   "HMI_DB".Drives.CU_U1.STW1.Bit00 := "DB_CU_U1".TelOut.CU_STW1.%X0;
   "HMI_DB".Drives.CU_U1.STW1.Bit01 := "DB_CU_U1".TelOut.CU_STW1.%X1;
   "HMI_DB".Drives.CU_U1.STW1.Bit02 := "DB_CU_U1".TelOut.CU_STW1.%X2;
   "HMI_DB".Drives.CU_U1.STW1.Bit03 := "DB_CU_U1".TelOut.CU_STW1.%X3;
   "HMI_DB".Drives.CU_U1.STW1.Bit04 := "DB_CU_U1".TelOut.CU_STW1.%X4;
   "HMI_DB".Drives.CU_U1.STW1.Bit05 := "DB_CU_U1".TelOut.CU_STW1.%X5;
   "HMI_DB".Drives.CU_U1.STW1.Bit06 := "DB_CU_U1".TelOut.CU_STW1.%X6;
   "HMI_DB".Drives.CU_U1.STW1.FaultAcknowledge := "DB_CU_U1".TelOut.CU_STW1.%X7;
   "HMI_DB".Drives.CU_U1.STW1.Bit08 := "DB_CU_U1".TelOut.CU_STW1.%X8;
   "HMI_DB".Drives.CU_U1.STW1.Bit09 := "DB_CU_U1".TelOut.CU_STW1.%X9;
   "HMI_DB".Drives.CU_U1.STW1.RemoteControlByPLC := "DB_CU_U1".TelOut.CU_STW1.%X10;
   "HMI_DB".Drives.CU_U1.STW1.Bit11 := "DB_CU_U1".TelOut.CU_STW1.%X11;
   "HMI_DB".Drives.CU_U1.STW1.Bit12 := "DB_CU_U1".TelOut.CU_STW1.%X12;
   "HMI_DB".Drives.CU_U1.STW1.Bit13 := "DB_CU_U1".TelOut.CU_STW1.%X13;
   "HMI_DB".Drives.CU_U1.STW1.Bit14 := "DB_CU_U1".TelOut.CU_STW1.%X14;
   "HMI_DB".Drives.CU_U1.STW1.Bit15 := "DB_CU_U1".TelOut.CU_STW1.%X15;


   // ============================================================
   // 6. CU_ZSW1 bits, CU -> PLC
   // ============================================================

   "HMI_DB".Drives.CU_U1.ZSW1.ReadyToSwitchOn := "DB_CU_U1".TelIn.CU_ZSW1.%X0;
   "HMI_DB".Drives.CU_U1.ZSW1.ReadyToOperate := "DB_CU_U1".TelIn.CU_ZSW1.%X1;
   "HMI_DB".Drives.CU_U1.ZSW1.OperationEnabled := "DB_CU_U1".TelIn.CU_ZSW1.%X2;
   "HMI_DB".Drives.CU_U1.ZSW1.FaultActive := "DB_CU_U1".TelIn.CU_ZSW1.%X3;
   "HMI_DB".Drives.CU_U1.ZSW1.NoCoastStopActive := "DB_CU_U1".TelIn.CU_ZSW1.%X4;
   "HMI_DB".Drives.CU_U1.ZSW1.NoQuickStopActive := "DB_CU_U1".TelIn.CU_ZSW1.%X5;
   "HMI_DB".Drives.CU_U1.ZSW1.SwitchingOnInhibit := "DB_CU_U1".TelIn.CU_ZSW1.%X6;
   "HMI_DB".Drives.CU_U1.ZSW1.WarningActive := "DB_CU_U1".TelIn.CU_ZSW1.%X7;
   "HMI_DB".Drives.CU_U1.ZSW1.Bit08 := "DB_CU_U1".TelIn.CU_ZSW1.%X8;
   "HMI_DB".Drives.CU_U1.ZSW1.ControlRequested := "DB_CU_U1".TelIn.CU_ZSW1.%X9;
   "HMI_DB".Drives.CU_U1.ZSW1.Bit10 := "DB_CU_U1".TelIn.CU_ZSW1.%X10;
   "HMI_DB".Drives.CU_U1.ZSW1.Bit11 := "DB_CU_U1".TelIn.CU_ZSW1.%X11;
   "HMI_DB".Drives.CU_U1.ZSW1.Bit12 := "DB_CU_U1".TelIn.CU_ZSW1.%X12;
   "HMI_DB".Drives.CU_U1.ZSW1.Bit13 := "DB_CU_U1".TelIn.CU_ZSW1.%X13;
   "HMI_DB".Drives.CU_U1.ZSW1.Bit14 := "DB_CU_U1".TelIn.CU_ZSW1.%X14;
   "HMI_DB".Drives.CU_U1.ZSW1.Bit15 := "DB_CU_U1".TelIn.CU_ZSW1.%X15;
END_REGION
END_FUNCTION

FUNCTION "FC_Drives_HMI_Alarms" : Void   // FC53, LAD
TITLE = Формування слів аварій (Faults) ПЧ для HMI
{ S7_Optimized_Access := 'TRUE' }
VERSION : 0.1
BEGIN

REGION Network 2 (SCL): Формування слів аварій для HMI - ПЧ 1UZ1
   // ============================================================
   // 1. FaultsWord1
   // ============================================================

   "HMI_DB".Drives.Drive_1UZ1.Faults.FaultsWord1.%X0 := "DB_Drive_1UZ1".Status.%X4 AND ("DB_Drive_1UZ1".FaultCode = W#16#03E8); // F01000
   "HMI_DB".Drives.Drive_1UZ1.Faults.FaultsWord1.%X1 := "DB_Drive_1UZ1".Status.%X4 AND ("DB_Drive_1UZ1".FaultCode = W#16#03E9); // F01001
   "HMI_DB".Drives.Drive_1UZ1.Faults.FaultsWord1.%X2 := "DB_Drive_1UZ1".Status.%X4 AND ("DB_Drive_1UZ1".FaultCode = W#16#03F7); // F01015
   "HMI_DB".Drives.Drive_1UZ1.Faults.FaultsWord1.%X3 := "DB_Drive_1UZ1".Status.%X4 AND ("DB_Drive_1UZ1".FaultCode = W#16#0409); // F01033
   "HMI_DB".Drives.Drive_1UZ1.Faults.FaultsWord1.%X4 := "DB_Drive_1UZ1".Status.%X4 AND ("DB_Drive_1UZ1".FaultCode = W#16#040A); // F01034
   "HMI_DB".Drives.Drive_1UZ1.Faults.FaultsWord1.%X5 := "DB_Drive_1UZ1".Status.%X4 AND ("DB_Drive_1UZ1".FaultCode = W#16#0410); // F01040
   "HMI_DB".Drives.Drive_1UZ1.Faults.FaultsWord1.%X6 := "DB_Drive_1UZ1".Status.%X4 AND ("DB_Drive_1UZ1".FaultCode = W#16#0414); // F01044
   "HMI_DB".Drives.Drive_1UZ1.Faults.FaultsWord1.%X7 := "DB_Drive_1UZ1".Status.%X4 AND ("DB_Drive_1UZ1".FaultCode = W#16#041E); // F01054
   "HMI_DB".Drives.Drive_1UZ1.Faults.FaultsWord1.%X8 := "DB_Drive_1UZ1".Status.%X4 AND ("DB_Drive_1UZ1".FaultCode = W#16#0451); // F01105
   "HMI_DB".Drives.Drive_1UZ1.Faults.FaultsWord1.%X9 := "DB_Drive_1UZ1".Status.%X4 AND ("DB_Drive_1UZ1".FaultCode = W#16#0462); // F01122
   "HMI_DB".Drives.Drive_1UZ1.Faults.FaultsWord1.%X10 := "DB_Drive_1UZ1".Status.%X4 AND ("DB_Drive_1UZ1".FaultCode = W#16#04B5); // F01205
   "HMI_DB".Drives.Drive_1UZ1.Faults.FaultsWord1.%X11 := "DB_Drive_1UZ1".Status.%X4 AND ("DB_Drive_1UZ1".FaultCode = W#16#04E2); // F01250
   "HMI_DB".Drives.Drive_1UZ1.Faults.FaultsWord1.%X12 := "DB_Drive_1UZ1".Status.%X4 AND ("DB_Drive_1UZ1".FaultCode = W#16#05E8); // F01512
   "HMI_DB".Drives.Drive_1UZ1.Faults.FaultsWord1.%X13 := "DB_Drive_1UZ1".Status.%X4 AND ("DB_Drive_1UZ1".FaultCode = W#16#0640); // F01600
   "HMI_DB".Drives.Drive_1UZ1.Faults.FaultsWord1.%X14 := "DB_Drive_1UZ1".Status.%X4 AND ("DB_Drive_1UZ1".FaultCode = W#16#0659); // F01625
   "HMI_DB".Drives.Drive_1UZ1.Faults.FaultsWord1.%X15 := "DB_Drive_1UZ1".Status.%X4 AND ("DB_Drive_1UZ1".FaultCode = W#16#0672); // F01650


   // ============================================================
   // 2. FaultsWord2
   // ============================================================

   "HMI_DB".Drives.Drive_1UZ1.Faults.FaultsWord2.%X0 := "DB_Drive_1UZ1".Status.%X4 AND ("DB_Drive_1UZ1".FaultCode = W#16#067B); // F01659
   "HMI_DB".Drives.Drive_1UZ1.Faults.FaultsWord2.%X1 := "DB_Drive_1UZ1".Status.%X4 AND ("DB_Drive_1UZ1".FaultCode = W#16#0682); // F01666
   "HMI_DB".Drives.Drive_1UZ1.Faults.FaultsWord2.%X2 := "DB_Drive_1UZ1".Status.%X4 AND ("DB_Drive_1UZ1".FaultCode = W#16#0776); // F01910
   "HMI_DB".Drives.Drive_1UZ1.Faults.FaultsWord2.%X3 := "DB_Drive_1UZ1".Status.%X4 AND ("DB_Drive_1UZ1".FaultCode = W#16#18A6); // F06310
   "HMI_DB".Drives.Drive_1UZ1.Faults.FaultsWord2.%X4 := "DB_Drive_1UZ1".Status.%X4 AND ("DB_Drive_1UZ1".FaultCode = W#16#1B63); // F07011
   "HMI_DB".Drives.Drive_1UZ1.Faults.FaultsWord2.%X5 := "DB_Drive_1UZ1".Status.%X4 AND ("DB_Drive_1UZ1".FaultCode = W#16#1B68); // F07016
   "HMI_DB".Drives.Drive_1UZ1.Faults.FaultsWord2.%X6 := "DB_Drive_1UZ1".Status.%X4 AND ("DB_Drive_1UZ1".FaultCode = W#16#1BAE); // F07086
   "HMI_DB".Drives.Drive_1UZ1.Faults.FaultsWord2.%X7 := "DB_Drive_1UZ1".Status.%X4 AND ("DB_Drive_1UZ1".FaultCode = W#16#1BB0); // F07088
   "HMI_DB".Drives.Drive_1UZ1.Faults.FaultsWord2.%X8 := "DB_Drive_1UZ1".Status.%X4 AND ("DB_Drive_1UZ1".FaultCode = W#16#1C98); // F07320
   "HMI_DB".Drives.Drive_1UZ1.Faults.FaultsWord2.%X9 := "DB_Drive_1UZ1".Status.%X4 AND ("DB_Drive_1UZ1".FaultCode = W#16#1CA2); // F07330
   "HMI_DB".Drives.Drive_1UZ1.Faults.FaultsWord2.%X10 := "DB_Drive_1UZ1".Status.%X4 AND ("DB_Drive_1UZ1".FaultCode = W#16#1D02); // F07426
   "HMI_DB".Drives.Drive_1UZ1.Faults.FaultsWord2.%X11 := "DB_Drive_1UZ1".Status.%X4 AND ("DB_Drive_1UZ1".FaultCode = W#16#1E79); // F07801
   "HMI_DB".Drives.Drive_1UZ1.Faults.FaultsWord2.%X12 := "DB_Drive_1UZ1".Status.%X4 AND ("DB_Drive_1UZ1".FaultCode = W#16#1E7F); // F07807
   "HMI_DB".Drives.Drive_1UZ1.Faults.FaultsWord2.%X13 := "DB_Drive_1UZ1".Status.%X4 AND ("DB_Drive_1UZ1".FaultCode = W#16#1EB4); // F07860
   "HMI_DB".Drives.Drive_1UZ1.Faults.FaultsWord2.%X14 := "DB_Drive_1UZ1".Status.%X4 AND ("DB_Drive_1UZ1".FaultCode = W#16#1EB5); // F07861
   "HMI_DB".Drives.Drive_1UZ1.Faults.FaultsWord2.%X15 := "DB_Drive_1UZ1".Status.%X4 AND ("DB_Drive_1UZ1".FaultCode = W#16#1EB6); // F07862


   // ============================================================
   // 3. FaultsWord3
   // ============================================================

   "HMI_DB".Drives.Drive_1UZ1.Faults.FaultsWord3.%X0 := "DB_Drive_1UZ1".Status.%X4 AND ("DB_Drive_1UZ1".FaultCode = W#16#1EDC); // F07900
   "HMI_DB".Drives.Drive_1UZ1.Faults.FaultsWord3.%X1 := "DB_Drive_1UZ1".Status.%X4 AND ("DB_Drive_1UZ1".FaultCode = W#16#1EDD); // F07901
   "HMI_DB".Drives.Drive_1UZ1.Faults.FaultsWord3.%X2 := "DB_Drive_1UZ1".Status.%X4 AND ("DB_Drive_1UZ1".FaultCode = W#16#1EDE); // F07902
   "HMI_DB".Drives.Drive_1UZ1.Faults.FaultsWord3.%X3 := "DB_Drive_1UZ1".Status.%X4 AND ("DB_Drive_1UZ1".FaultCode = W#16#1EF3); // F07923
   "HMI_DB".Drives.Drive_1UZ1.Faults.FaultsWord3.%X4 := "DB_Drive_1UZ1".Status.%X4 AND ("DB_Drive_1UZ1".FaultCode = W#16#1EF4); // F07924
   "HMI_DB".Drives.Drive_1UZ1.Faults.FaultsWord3.%X5 := "DB_Drive_1UZ1".Status.%X4 AND ("DB_Drive_1UZ1".FaultCode = W#16#2135); // F08501
   "HMI_DB".Drives.Drive_1UZ1.Faults.FaultsWord3.%X6 := "DB_Drive_1UZ1".Status.%X4 AND ("DB_Drive_1UZ1".FaultCode = W#16#2136); // F08502
   "HMI_DB".Drives.Drive_1UZ1.Faults.FaultsWord3.%X7 := "DB_Drive_1UZ1".Status.%X4 AND ("DB_Drive_1UZ1".FaultCode = W#16#1842); // F06210
   "HMI_DB".Drives.Drive_1UZ1.Faults.FaultsWord3.%X8 := "DB_Drive_1UZ1".Status.%X4 AND ("DB_Drive_1UZ1".FaultCode = W#16#332C); // F13100
   "HMI_DB".Drives.Drive_1UZ1.Faults.FaultsWord3.%X9 := "DB_Drive_1UZ1".Status.%X4 AND ("DB_Drive_1UZ1".FaultCode = W#16#332D); // F13101
   "HMI_DB".Drives.Drive_1UZ1.Faults.FaultsWord3.%X10 := "DB_Drive_1UZ1".Status.%X4 AND ("DB_Drive_1UZ1".FaultCode = W#16#7531); // F30001
   "HMI_DB".Drives.Drive_1UZ1.Faults.FaultsWord3.%X11 := "DB_Drive_1UZ1".Status.%X4 AND ("DB_Drive_1UZ1".FaultCode = W#16#7532); // F30002
   "HMI_DB".Drives.Drive_1UZ1.Faults.FaultsWord3.%X12 := "DB_Drive_1UZ1".Status.%X4 AND ("DB_Drive_1UZ1".FaultCode = W#16#7533); // F30003
   "HMI_DB".Drives.Drive_1UZ1.Faults.FaultsWord3.%X13 := "DB_Drive_1UZ1".Status.%X4 AND ("DB_Drive_1UZ1".FaultCode = W#16#7534); // F30004
   "HMI_DB".Drives.Drive_1UZ1.Faults.FaultsWord3.%X14 := "DB_Drive_1UZ1".Status.%X4 AND ("DB_Drive_1UZ1".FaultCode = W#16#7535); // F30005
   "HMI_DB".Drives.Drive_1UZ1.Faults.FaultsWord3.%X15 := "DB_Drive_1UZ1".Status.%X4 AND ("DB_Drive_1UZ1".FaultCode = W#16#753B); // F30011


   // ============================================================
   // 4. FaultsWord4
   // ============================================================

   "HMI_DB".Drives.Drive_1UZ1.Faults.FaultsWord4.%X0 := "DB_Drive_1UZ1".Status.%X4 AND ("DB_Drive_1UZ1".FaultCode = W#16#753F); // F30015
   "HMI_DB".Drives.Drive_1UZ1.Faults.FaultsWord4.%X1 := "DB_Drive_1UZ1".Status.%X4 AND ("DB_Drive_1UZ1".FaultCode = W#16#7545); // F30021
   "HMI_DB".Drives.Drive_1UZ1.Faults.FaultsWord4.%X2 := "DB_Drive_1UZ1".Status.%X4 AND ("DB_Drive_1UZ1".FaultCode = W#16#7546); // F30022
   "HMI_DB".Drives.Drive_1UZ1.Faults.FaultsWord4.%X3 := "DB_Drive_1UZ1".Status.%X4 AND ("DB_Drive_1UZ1".FaultCode = W#16#754B); // F30027
   "HMI_DB".Drives.Drive_1UZ1.Faults.FaultsWord4.%X4 := "DB_Drive_1UZ1".Status.%X4 AND ("DB_Drive_1UZ1".FaultCode = W#16#7553); // F30035
   "HMI_DB".Drives.Drive_1UZ1.Faults.FaultsWord4.%X5 := "DB_Drive_1UZ1".Status.%X4 AND ("DB_Drive_1UZ1".FaultCode = W#16#7554); // F30036
   "HMI_DB".Drives.Drive_1UZ1.Faults.FaultsWord4.%X6 := "DB_Drive_1UZ1".Status.%X4 AND ("DB_Drive_1UZ1".FaultCode = W#16#7555); // F30037
   "HMI_DB".Drives.Drive_1UZ1.Faults.FaultsWord4.%X7 := "DB_Drive_1UZ1".Status.%X4 AND ("DB_Drive_1UZ1".FaultCode = W#16#7564); // F30052
   "HMI_DB".Drives.Drive_1UZ1.Faults.FaultsWord4.%X8 := "DB_Drive_1UZ1".Status.%X4 AND ("DB_Drive_1UZ1".FaultCode = W#16#7565); // F30053
   "HMI_DB".Drives.Drive_1UZ1.Faults.FaultsWord4.%X9 := "DB_Drive_1UZ1".Status.%X4 AND ("DB_Drive_1UZ1".FaultCode = W#16#756B); // F30059
   "HMI_DB".Drives.Drive_1UZ1.Faults.FaultsWord4.%X10 := "DB_Drive_1UZ1".Status.%X4 AND ("DB_Drive_1UZ1".FaultCode = W#16#757A); // F30074
   "HMI_DB".Drives.Drive_1UZ1.Faults.FaultsWord4.%X11 := "DB_Drive_1UZ1".Status.%X4 AND ("DB_Drive_1UZ1".FaultCode = W#16#7788); // F30600
   "HMI_DB".Drives.Drive_1UZ1.Faults.FaultsWord4.%X12 := "DB_Drive_1UZ1".Status.%X4 AND ("DB_Drive_1UZ1".FaultCode = W#16#77C8); // F30664
   "HMI_DB".Drives.Drive_1UZ1.Faults.FaultsWord4.%X13 := "DB_Drive_1UZ1".Status.%X4 AND ("DB_Drive_1UZ1".FaultCode = W#16#7882); // F30850
   "HMI_DB".Drives.Drive_1UZ1.Faults.FaultsWord4.%X14 := "DB_Drive_1UZ1".Status.%X4 AND ("DB_Drive_1UZ1".FaultCode = W#16#1843); // F06211
   "HMI_DB".Drives.Drive_1UZ1.Faults.FaultsWord4.%X15 := "DB_Drive_1UZ1".Status.%X4 AND ("DB_Drive_1UZ1".FaultCode = W#16#213E); // F08510
END_REGION

REGION Network 3 (SCL): Формування слів аварій для HMI - ПЧ 3UZ1
   // ============================================================
   // 1. FaultsWord1
   // ============================================================

   "HMI_DB".Drives.Drive_3UZ1.Faults.FaultsWord1.%X0 := "DB_Drive_3UZ1".Status.%X4 AND ("DB_Drive_3UZ1".FaultCode = W#16#03E8); // F01000
   "HMI_DB".Drives.Drive_3UZ1.Faults.FaultsWord1.%X1 := "DB_Drive_3UZ1".Status.%X4 AND ("DB_Drive_3UZ1".FaultCode = W#16#03E9); // F01001
   "HMI_DB".Drives.Drive_3UZ1.Faults.FaultsWord1.%X2 := "DB_Drive_3UZ1".Status.%X4 AND ("DB_Drive_3UZ1".FaultCode = W#16#03F7); // F01015
   "HMI_DB".Drives.Drive_3UZ1.Faults.FaultsWord1.%X3 := "DB_Drive_3UZ1".Status.%X4 AND ("DB_Drive_3UZ1".FaultCode = W#16#0409); // F01033
   "HMI_DB".Drives.Drive_3UZ1.Faults.FaultsWord1.%X4 := "DB_Drive_3UZ1".Status.%X4 AND ("DB_Drive_3UZ1".FaultCode = W#16#040A); // F01034
   "HMI_DB".Drives.Drive_3UZ1.Faults.FaultsWord1.%X5 := "DB_Drive_3UZ1".Status.%X4 AND ("DB_Drive_3UZ1".FaultCode = W#16#0410); // F01040
   "HMI_DB".Drives.Drive_3UZ1.Faults.FaultsWord1.%X6 := "DB_Drive_3UZ1".Status.%X4 AND ("DB_Drive_3UZ1".FaultCode = W#16#0414); // F01044
   "HMI_DB".Drives.Drive_3UZ1.Faults.FaultsWord1.%X7 := "DB_Drive_3UZ1".Status.%X4 AND ("DB_Drive_3UZ1".FaultCode = W#16#041E); // F01054
   "HMI_DB".Drives.Drive_3UZ1.Faults.FaultsWord1.%X8 := "DB_Drive_3UZ1".Status.%X4 AND ("DB_Drive_3UZ1".FaultCode = W#16#0451); // F01105
   "HMI_DB".Drives.Drive_3UZ1.Faults.FaultsWord1.%X9 := "DB_Drive_3UZ1".Status.%X4 AND ("DB_Drive_3UZ1".FaultCode = W#16#0462); // F01122
   "HMI_DB".Drives.Drive_3UZ1.Faults.FaultsWord1.%X10 := "DB_Drive_3UZ1".Status.%X4 AND ("DB_Drive_3UZ1".FaultCode = W#16#04B5); // F01205
   "HMI_DB".Drives.Drive_3UZ1.Faults.FaultsWord1.%X11 := "DB_Drive_3UZ1".Status.%X4 AND ("DB_Drive_3UZ1".FaultCode = W#16#04E2); // F01250
   "HMI_DB".Drives.Drive_3UZ1.Faults.FaultsWord1.%X12 := "DB_Drive_3UZ1".Status.%X4 AND ("DB_Drive_3UZ1".FaultCode = W#16#05E8); // F01512
   "HMI_DB".Drives.Drive_3UZ1.Faults.FaultsWord1.%X13 := "DB_Drive_3UZ1".Status.%X4 AND ("DB_Drive_3UZ1".FaultCode = W#16#0640); // F01600
   "HMI_DB".Drives.Drive_3UZ1.Faults.FaultsWord1.%X14 := "DB_Drive_3UZ1".Status.%X4 AND ("DB_Drive_3UZ1".FaultCode = W#16#0659); // F01625
   "HMI_DB".Drives.Drive_3UZ1.Faults.FaultsWord1.%X15 := "DB_Drive_3UZ1".Status.%X4 AND ("DB_Drive_3UZ1".FaultCode = W#16#0672); // F01650


   // ============================================================
   // 2. FaultsWord2
   // ============================================================

   "HMI_DB".Drives.Drive_3UZ1.Faults.FaultsWord2.%X0 := "DB_Drive_3UZ1".Status.%X4 AND ("DB_Drive_3UZ1".FaultCode = W#16#067B); // F01659
   "HMI_DB".Drives.Drive_3UZ1.Faults.FaultsWord2.%X1 := "DB_Drive_3UZ1".Status.%X4 AND ("DB_Drive_3UZ1".FaultCode = W#16#0682); // F01666
   "HMI_DB".Drives.Drive_3UZ1.Faults.FaultsWord2.%X2 := "DB_Drive_3UZ1".Status.%X4 AND ("DB_Drive_3UZ1".FaultCode = W#16#0776); // F01910
   "HMI_DB".Drives.Drive_3UZ1.Faults.FaultsWord2.%X3 := "DB_Drive_3UZ1".Status.%X4 AND ("DB_Drive_3UZ1".FaultCode = W#16#18A6); // F06310
   "HMI_DB".Drives.Drive_3UZ1.Faults.FaultsWord2.%X4 := "DB_Drive_3UZ1".Status.%X4 AND ("DB_Drive_3UZ1".FaultCode = W#16#1B63); // F07011
   "HMI_DB".Drives.Drive_3UZ1.Faults.FaultsWord2.%X5 := "DB_Drive_3UZ1".Status.%X4 AND ("DB_Drive_3UZ1".FaultCode = W#16#1B68); // F07016
   "HMI_DB".Drives.Drive_3UZ1.Faults.FaultsWord2.%X6 := "DB_Drive_3UZ1".Status.%X4 AND ("DB_Drive_3UZ1".FaultCode = W#16#1BAE); // F07086
   "HMI_DB".Drives.Drive_3UZ1.Faults.FaultsWord2.%X7 := "DB_Drive_3UZ1".Status.%X4 AND ("DB_Drive_3UZ1".FaultCode = W#16#1BB0); // F07088
   "HMI_DB".Drives.Drive_3UZ1.Faults.FaultsWord2.%X8 := "DB_Drive_3UZ1".Status.%X4 AND ("DB_Drive_3UZ1".FaultCode = W#16#1C98); // F07320
   "HMI_DB".Drives.Drive_3UZ1.Faults.FaultsWord2.%X9 := "DB_Drive_3UZ1".Status.%X4 AND ("DB_Drive_3UZ1".FaultCode = W#16#1CA2); // F07330
   "HMI_DB".Drives.Drive_3UZ1.Faults.FaultsWord2.%X10 := "DB_Drive_3UZ1".Status.%X4 AND ("DB_Drive_3UZ1".FaultCode = W#16#1D02); // F07426
   "HMI_DB".Drives.Drive_3UZ1.Faults.FaultsWord2.%X11 := "DB_Drive_3UZ1".Status.%X4 AND ("DB_Drive_3UZ1".FaultCode = W#16#1E79); // F07801
   "HMI_DB".Drives.Drive_3UZ1.Faults.FaultsWord2.%X12 := "DB_Drive_3UZ1".Status.%X4 AND ("DB_Drive_3UZ1".FaultCode = W#16#1E7F); // F07807
   "HMI_DB".Drives.Drive_3UZ1.Faults.FaultsWord2.%X13 := "DB_Drive_3UZ1".Status.%X4 AND ("DB_Drive_3UZ1".FaultCode = W#16#1EB4); // F07860
   "HMI_DB".Drives.Drive_3UZ1.Faults.FaultsWord2.%X14 := "DB_Drive_3UZ1".Status.%X4 AND ("DB_Drive_3UZ1".FaultCode = W#16#1EB5); // F07861
   "HMI_DB".Drives.Drive_3UZ1.Faults.FaultsWord2.%X15 := "DB_Drive_3UZ1".Status.%X4 AND ("DB_Drive_3UZ1".FaultCode = W#16#1EB6); // F07862


   // ============================================================
   // 3. FaultsWord3
   // ============================================================

   "HMI_DB".Drives.Drive_3UZ1.Faults.FaultsWord3.%X0 := "DB_Drive_3UZ1".Status.%X4 AND ("DB_Drive_3UZ1".FaultCode = W#16#1EDC); // F07900
   "HMI_DB".Drives.Drive_3UZ1.Faults.FaultsWord3.%X1 := "DB_Drive_3UZ1".Status.%X4 AND ("DB_Drive_3UZ1".FaultCode = W#16#1EDD); // F07901
   "HMI_DB".Drives.Drive_3UZ1.Faults.FaultsWord3.%X2 := "DB_Drive_3UZ1".Status.%X4 AND ("DB_Drive_3UZ1".FaultCode = W#16#1EDE); // F07902
   "HMI_DB".Drives.Drive_3UZ1.Faults.FaultsWord3.%X3 := "DB_Drive_3UZ1".Status.%X4 AND ("DB_Drive_3UZ1".FaultCode = W#16#1EF3); // F07923
   "HMI_DB".Drives.Drive_3UZ1.Faults.FaultsWord3.%X4 := "DB_Drive_3UZ1".Status.%X4 AND ("DB_Drive_3UZ1".FaultCode = W#16#1EF4); // F07924
   "HMI_DB".Drives.Drive_3UZ1.Faults.FaultsWord3.%X5 := "DB_Drive_3UZ1".Status.%X4 AND ("DB_Drive_3UZ1".FaultCode = W#16#2135); // F08501
   "HMI_DB".Drives.Drive_3UZ1.Faults.FaultsWord3.%X6 := "DB_Drive_3UZ1".Status.%X4 AND ("DB_Drive_3UZ1".FaultCode = W#16#2136); // F08502
   "HMI_DB".Drives.Drive_3UZ1.Faults.FaultsWord3.%X7 := "DB_Drive_3UZ1".Status.%X4 AND ("DB_Drive_3UZ1".FaultCode = W#16#1842); // F06210
   "HMI_DB".Drives.Drive_3UZ1.Faults.FaultsWord3.%X8 := "DB_Drive_3UZ1".Status.%X4 AND ("DB_Drive_3UZ1".FaultCode = W#16#332C); // F13100
   "HMI_DB".Drives.Drive_3UZ1.Faults.FaultsWord3.%X9 := "DB_Drive_3UZ1".Status.%X4 AND ("DB_Drive_3UZ1".FaultCode = W#16#332D); // F13101
   "HMI_DB".Drives.Drive_3UZ1.Faults.FaultsWord3.%X10 := "DB_Drive_3UZ1".Status.%X4 AND ("DB_Drive_3UZ1".FaultCode = W#16#7531); // F30001
   "HMI_DB".Drives.Drive_3UZ1.Faults.FaultsWord3.%X11 := "DB_Drive_3UZ1".Status.%X4 AND ("DB_Drive_3UZ1".FaultCode = W#16#7532); // F30002
   "HMI_DB".Drives.Drive_3UZ1.Faults.FaultsWord3.%X12 := "DB_Drive_3UZ1".Status.%X4 AND ("DB_Drive_3UZ1".FaultCode = W#16#7533); // F30003
   "HMI_DB".Drives.Drive_3UZ1.Faults.FaultsWord3.%X13 := "DB_Drive_3UZ1".Status.%X4 AND ("DB_Drive_3UZ1".FaultCode = W#16#7534); // F30004
   "HMI_DB".Drives.Drive_3UZ1.Faults.FaultsWord3.%X14 := "DB_Drive_3UZ1".Status.%X4 AND ("DB_Drive_3UZ1".FaultCode = W#16#7535); // F30005
   "HMI_DB".Drives.Drive_3UZ1.Faults.FaultsWord3.%X15 := "DB_Drive_3UZ1".Status.%X4 AND ("DB_Drive_3UZ1".FaultCode = W#16#753B); // F30011


   // ============================================================
   // 4. FaultsWord4
   // ============================================================

   "HMI_DB".Drives.Drive_3UZ1.Faults.FaultsWord4.%X0 := "DB_Drive_3UZ1".Status.%X4 AND ("DB_Drive_3UZ1".FaultCode = W#16#753F); // F30015
   "HMI_DB".Drives.Drive_3UZ1.Faults.FaultsWord4.%X1 := "DB_Drive_3UZ1".Status.%X4 AND ("DB_Drive_3UZ1".FaultCode = W#16#7545); // F30021
   "HMI_DB".Drives.Drive_3UZ1.Faults.FaultsWord4.%X2 := "DB_Drive_3UZ1".Status.%X4 AND ("DB_Drive_3UZ1".FaultCode = W#16#7546); // F30022
   "HMI_DB".Drives.Drive_3UZ1.Faults.FaultsWord4.%X3 := "DB_Drive_3UZ1".Status.%X4 AND ("DB_Drive_3UZ1".FaultCode = W#16#754B); // F30027
   "HMI_DB".Drives.Drive_3UZ1.Faults.FaultsWord4.%X4 := "DB_Drive_3UZ1".Status.%X4 AND ("DB_Drive_3UZ1".FaultCode = W#16#7553); // F30035
   "HMI_DB".Drives.Drive_3UZ1.Faults.FaultsWord4.%X5 := "DB_Drive_3UZ1".Status.%X4 AND ("DB_Drive_3UZ1".FaultCode = W#16#7554); // F30036
   "HMI_DB".Drives.Drive_3UZ1.Faults.FaultsWord4.%X6 := "DB_Drive_3UZ1".Status.%X4 AND ("DB_Drive_3UZ1".FaultCode = W#16#7555); // F30037
   "HMI_DB".Drives.Drive_3UZ1.Faults.FaultsWord4.%X7 := "DB_Drive_3UZ1".Status.%X4 AND ("DB_Drive_3UZ1".FaultCode = W#16#7564); // F30052
   "HMI_DB".Drives.Drive_3UZ1.Faults.FaultsWord4.%X8 := "DB_Drive_3UZ1".Status.%X4 AND ("DB_Drive_3UZ1".FaultCode = W#16#7565); // F30053
   "HMI_DB".Drives.Drive_3UZ1.Faults.FaultsWord4.%X9 := "DB_Drive_3UZ1".Status.%X4 AND ("DB_Drive_3UZ1".FaultCode = W#16#756B); // F30059
   "HMI_DB".Drives.Drive_3UZ1.Faults.FaultsWord4.%X10 := "DB_Drive_3UZ1".Status.%X4 AND ("DB_Drive_3UZ1".FaultCode = W#16#757A); // F30074
   "HMI_DB".Drives.Drive_3UZ1.Faults.FaultsWord4.%X11 := "DB_Drive_3UZ1".Status.%X4 AND ("DB_Drive_3UZ1".FaultCode = W#16#7788); // F30600
   "HMI_DB".Drives.Drive_3UZ1.Faults.FaultsWord4.%X12 := "DB_Drive_3UZ1".Status.%X4 AND ("DB_Drive_3UZ1".FaultCode = W#16#77C8); // F30664
   "HMI_DB".Drives.Drive_3UZ1.Faults.FaultsWord4.%X13 := "DB_Drive_3UZ1".Status.%X4 AND ("DB_Drive_3UZ1".FaultCode = W#16#7882); // F30850
   "HMI_DB".Drives.Drive_3UZ1.Faults.FaultsWord4.%X14 := "DB_Drive_3UZ1".Status.%X4 AND ("DB_Drive_3UZ1".FaultCode = W#16#1843); // F06211
   "HMI_DB".Drives.Drive_3UZ1.Faults.FaultsWord4.%X15 := "DB_Drive_3UZ1".Status.%X4 AND ("DB_Drive_3UZ1".FaultCode = W#16#213E); // F08510
END_REGION

REGION Network 4 (SCL): Формування слів аварій для HMI - ПЧ 4UZ1
   // ============================================================
   // 1. FaultsWord1
   // ============================================================

   "HMI_DB".Drives.Drive_4UZ1.Faults.FaultsWord1.%X0 := "DB_Drive_4UZ1".Status.%X4 AND ("DB_Drive_4UZ1".FaultCode = W#16#03E8); // F01000
   "HMI_DB".Drives.Drive_4UZ1.Faults.FaultsWord1.%X1 := "DB_Drive_4UZ1".Status.%X4 AND ("DB_Drive_4UZ1".FaultCode = W#16#03E9); // F01001
   "HMI_DB".Drives.Drive_4UZ1.Faults.FaultsWord1.%X2 := "DB_Drive_4UZ1".Status.%X4 AND ("DB_Drive_4UZ1".FaultCode = W#16#03F7); // F01015
   "HMI_DB".Drives.Drive_4UZ1.Faults.FaultsWord1.%X3 := "DB_Drive_4UZ1".Status.%X4 AND ("DB_Drive_4UZ1".FaultCode = W#16#0409); // F01033
   "HMI_DB".Drives.Drive_4UZ1.Faults.FaultsWord1.%X4 := "DB_Drive_4UZ1".Status.%X4 AND ("DB_Drive_4UZ1".FaultCode = W#16#040A); // F01034
   "HMI_DB".Drives.Drive_4UZ1.Faults.FaultsWord1.%X5 := "DB_Drive_4UZ1".Status.%X4 AND ("DB_Drive_4UZ1".FaultCode = W#16#0410); // F01040
   "HMI_DB".Drives.Drive_4UZ1.Faults.FaultsWord1.%X6 := "DB_Drive_4UZ1".Status.%X4 AND ("DB_Drive_4UZ1".FaultCode = W#16#0414); // F01044
   "HMI_DB".Drives.Drive_4UZ1.Faults.FaultsWord1.%X7 := "DB_Drive_4UZ1".Status.%X4 AND ("DB_Drive_4UZ1".FaultCode = W#16#041E); // F01054
   "HMI_DB".Drives.Drive_4UZ1.Faults.FaultsWord1.%X8 := "DB_Drive_4UZ1".Status.%X4 AND ("DB_Drive_4UZ1".FaultCode = W#16#0451); // F01105
   "HMI_DB".Drives.Drive_4UZ1.Faults.FaultsWord1.%X9 := "DB_Drive_4UZ1".Status.%X4 AND ("DB_Drive_4UZ1".FaultCode = W#16#0462); // F01122
   "HMI_DB".Drives.Drive_4UZ1.Faults.FaultsWord1.%X10 := "DB_Drive_4UZ1".Status.%X4 AND ("DB_Drive_4UZ1".FaultCode = W#16#04B5); // F01205
   "HMI_DB".Drives.Drive_4UZ1.Faults.FaultsWord1.%X11 := "DB_Drive_4UZ1".Status.%X4 AND ("DB_Drive_4UZ1".FaultCode = W#16#04E2); // F01250
   "HMI_DB".Drives.Drive_4UZ1.Faults.FaultsWord1.%X12 := "DB_Drive_4UZ1".Status.%X4 AND ("DB_Drive_4UZ1".FaultCode = W#16#05E8); // F01512
   "HMI_DB".Drives.Drive_4UZ1.Faults.FaultsWord1.%X13 := "DB_Drive_4UZ1".Status.%X4 AND ("DB_Drive_4UZ1".FaultCode = W#16#0640); // F01600
   "HMI_DB".Drives.Drive_4UZ1.Faults.FaultsWord1.%X14 := "DB_Drive_4UZ1".Status.%X4 AND ("DB_Drive_4UZ1".FaultCode = W#16#0659); // F01625
   "HMI_DB".Drives.Drive_4UZ1.Faults.FaultsWord1.%X15 := "DB_Drive_4UZ1".Status.%X4 AND ("DB_Drive_4UZ1".FaultCode = W#16#0672); // F01650


   // ============================================================
   // 2. FaultsWord2
   // ============================================================

   "HMI_DB".Drives.Drive_4UZ1.Faults.FaultsWord2.%X0 := "DB_Drive_4UZ1".Status.%X4 AND ("DB_Drive_4UZ1".FaultCode = W#16#067B); // F01659
   "HMI_DB".Drives.Drive_4UZ1.Faults.FaultsWord2.%X1 := "DB_Drive_4UZ1".Status.%X4 AND ("DB_Drive_4UZ1".FaultCode = W#16#0682); // F01666
   "HMI_DB".Drives.Drive_4UZ1.Faults.FaultsWord2.%X2 := "DB_Drive_4UZ1".Status.%X4 AND ("DB_Drive_4UZ1".FaultCode = W#16#0776); // F01910
   "HMI_DB".Drives.Drive_4UZ1.Faults.FaultsWord2.%X3 := "DB_Drive_4UZ1".Status.%X4 AND ("DB_Drive_4UZ1".FaultCode = W#16#18A6); // F06310
   "HMI_DB".Drives.Drive_4UZ1.Faults.FaultsWord2.%X4 := "DB_Drive_4UZ1".Status.%X4 AND ("DB_Drive_4UZ1".FaultCode = W#16#1B63); // F07011
   "HMI_DB".Drives.Drive_4UZ1.Faults.FaultsWord2.%X5 := "DB_Drive_4UZ1".Status.%X4 AND ("DB_Drive_4UZ1".FaultCode = W#16#1B68); // F07016
   "HMI_DB".Drives.Drive_4UZ1.Faults.FaultsWord2.%X6 := "DB_Drive_4UZ1".Status.%X4 AND ("DB_Drive_4UZ1".FaultCode = W#16#1BAE); // F07086
   "HMI_DB".Drives.Drive_4UZ1.Faults.FaultsWord2.%X7 := "DB_Drive_4UZ1".Status.%X4 AND ("DB_Drive_4UZ1".FaultCode = W#16#1BB0); // F07088
   "HMI_DB".Drives.Drive_4UZ1.Faults.FaultsWord2.%X8 := "DB_Drive_4UZ1".Status.%X4 AND ("DB_Drive_4UZ1".FaultCode = W#16#1C98); // F07320
   "HMI_DB".Drives.Drive_4UZ1.Faults.FaultsWord2.%X9 := "DB_Drive_4UZ1".Status.%X4 AND ("DB_Drive_4UZ1".FaultCode = W#16#1CA2); // F07330
   "HMI_DB".Drives.Drive_4UZ1.Faults.FaultsWord2.%X10 := "DB_Drive_4UZ1".Status.%X4 AND ("DB_Drive_4UZ1".FaultCode = W#16#1D02); // F07426
   "HMI_DB".Drives.Drive_4UZ1.Faults.FaultsWord2.%X11 := "DB_Drive_4UZ1".Status.%X4 AND ("DB_Drive_4UZ1".FaultCode = W#16#1E79); // F07801
   "HMI_DB".Drives.Drive_4UZ1.Faults.FaultsWord2.%X12 := "DB_Drive_4UZ1".Status.%X4 AND ("DB_Drive_4UZ1".FaultCode = W#16#1E7F); // F07807
   "HMI_DB".Drives.Drive_4UZ1.Faults.FaultsWord2.%X13 := "DB_Drive_4UZ1".Status.%X4 AND ("DB_Drive_4UZ1".FaultCode = W#16#1EB4); // F07860
   "HMI_DB".Drives.Drive_4UZ1.Faults.FaultsWord2.%X14 := "DB_Drive_4UZ1".Status.%X4 AND ("DB_Drive_4UZ1".FaultCode = W#16#1EB5); // F07861
   "HMI_DB".Drives.Drive_4UZ1.Faults.FaultsWord2.%X15 := "DB_Drive_4UZ1".Status.%X4 AND ("DB_Drive_4UZ1".FaultCode = W#16#1EB6); // F07862


   // ============================================================
   // 3. FaultsWord3
   // ============================================================

   "HMI_DB".Drives.Drive_4UZ1.Faults.FaultsWord3.%X0 := "DB_Drive_4UZ1".Status.%X4 AND ("DB_Drive_4UZ1".FaultCode = W#16#1EDC); // F07900
   "HMI_DB".Drives.Drive_4UZ1.Faults.FaultsWord3.%X1 := "DB_Drive_4UZ1".Status.%X4 AND ("DB_Drive_4UZ1".FaultCode = W#16#1EDD); // F07901
   "HMI_DB".Drives.Drive_4UZ1.Faults.FaultsWord3.%X2 := "DB_Drive_4UZ1".Status.%X4 AND ("DB_Drive_4UZ1".FaultCode = W#16#1EDE); // F07902
   "HMI_DB".Drives.Drive_4UZ1.Faults.FaultsWord3.%X3 := "DB_Drive_4UZ1".Status.%X4 AND ("DB_Drive_4UZ1".FaultCode = W#16#1EF3); // F07923
   "HMI_DB".Drives.Drive_4UZ1.Faults.FaultsWord3.%X4 := "DB_Drive_4UZ1".Status.%X4 AND ("DB_Drive_4UZ1".FaultCode = W#16#1EF4); // F07924
   "HMI_DB".Drives.Drive_4UZ1.Faults.FaultsWord3.%X5 := "DB_Drive_4UZ1".Status.%X4 AND ("DB_Drive_4UZ1".FaultCode = W#16#2135); // F08501
   "HMI_DB".Drives.Drive_4UZ1.Faults.FaultsWord3.%X6 := "DB_Drive_4UZ1".Status.%X4 AND ("DB_Drive_4UZ1".FaultCode = W#16#2136); // F08502
   "HMI_DB".Drives.Drive_4UZ1.Faults.FaultsWord3.%X7 := "DB_Drive_4UZ1".Status.%X4 AND ("DB_Drive_4UZ1".FaultCode = W#16#1842); // F06210
   "HMI_DB".Drives.Drive_4UZ1.Faults.FaultsWord3.%X8 := "DB_Drive_4UZ1".Status.%X4 AND ("DB_Drive_4UZ1".FaultCode = W#16#332C); // F13100
   "HMI_DB".Drives.Drive_4UZ1.Faults.FaultsWord3.%X9 := "DB_Drive_4UZ1".Status.%X4 AND ("DB_Drive_4UZ1".FaultCode = W#16#332D); // F13101
   "HMI_DB".Drives.Drive_4UZ1.Faults.FaultsWord3.%X10 := "DB_Drive_4UZ1".Status.%X4 AND ("DB_Drive_4UZ1".FaultCode = W#16#7531); // F30001
   "HMI_DB".Drives.Drive_4UZ1.Faults.FaultsWord3.%X11 := "DB_Drive_4UZ1".Status.%X4 AND ("DB_Drive_4UZ1".FaultCode = W#16#7532); // F30002
   "HMI_DB".Drives.Drive_4UZ1.Faults.FaultsWord3.%X12 := "DB_Drive_4UZ1".Status.%X4 AND ("DB_Drive_4UZ1".FaultCode = W#16#7533); // F30003
   "HMI_DB".Drives.Drive_4UZ1.Faults.FaultsWord3.%X13 := "DB_Drive_4UZ1".Status.%X4 AND ("DB_Drive_4UZ1".FaultCode = W#16#7534); // F30004
   "HMI_DB".Drives.Drive_4UZ1.Faults.FaultsWord3.%X14 := "DB_Drive_4UZ1".Status.%X4 AND ("DB_Drive_4UZ1".FaultCode = W#16#7535); // F30005
   "HMI_DB".Drives.Drive_4UZ1.Faults.FaultsWord3.%X15 := "DB_Drive_4UZ1".Status.%X4 AND ("DB_Drive_4UZ1".FaultCode = W#16#753B); // F30011


   // ============================================================
   // 4. FaultsWord4
   // ============================================================

   "HMI_DB".Drives.Drive_4UZ1.Faults.FaultsWord4.%X0 := "DB_Drive_4UZ1".Status.%X4 AND ("DB_Drive_4UZ1".FaultCode = W#16#753F); // F30015
   "HMI_DB".Drives.Drive_4UZ1.Faults.FaultsWord4.%X1 := "DB_Drive_4UZ1".Status.%X4 AND ("DB_Drive_4UZ1".FaultCode = W#16#7545); // F30021
   "HMI_DB".Drives.Drive_4UZ1.Faults.FaultsWord4.%X2 := "DB_Drive_4UZ1".Status.%X4 AND ("DB_Drive_4UZ1".FaultCode = W#16#7546); // F30022
   "HMI_DB".Drives.Drive_4UZ1.Faults.FaultsWord4.%X3 := "DB_Drive_4UZ1".Status.%X4 AND ("DB_Drive_4UZ1".FaultCode = W#16#754B); // F30027
   "HMI_DB".Drives.Drive_4UZ1.Faults.FaultsWord4.%X4 := "DB_Drive_4UZ1".Status.%X4 AND ("DB_Drive_4UZ1".FaultCode = W#16#7553); // F30035
   "HMI_DB".Drives.Drive_4UZ1.Faults.FaultsWord4.%X5 := "DB_Drive_4UZ1".Status.%X4 AND ("DB_Drive_4UZ1".FaultCode = W#16#7554); // F30036
   "HMI_DB".Drives.Drive_4UZ1.Faults.FaultsWord4.%X6 := "DB_Drive_4UZ1".Status.%X4 AND ("DB_Drive_4UZ1".FaultCode = W#16#7555); // F30037
   "HMI_DB".Drives.Drive_4UZ1.Faults.FaultsWord4.%X7 := "DB_Drive_4UZ1".Status.%X4 AND ("DB_Drive_4UZ1".FaultCode = W#16#7564); // F30052
   "HMI_DB".Drives.Drive_4UZ1.Faults.FaultsWord4.%X8 := "DB_Drive_4UZ1".Status.%X4 AND ("DB_Drive_4UZ1".FaultCode = W#16#7565); // F30053
   "HMI_DB".Drives.Drive_4UZ1.Faults.FaultsWord4.%X9 := "DB_Drive_4UZ1".Status.%X4 AND ("DB_Drive_4UZ1".FaultCode = W#16#756B); // F30059
   "HMI_DB".Drives.Drive_4UZ1.Faults.FaultsWord4.%X10 := "DB_Drive_4UZ1".Status.%X4 AND ("DB_Drive_4UZ1".FaultCode = W#16#757A); // F30074
   "HMI_DB".Drives.Drive_4UZ1.Faults.FaultsWord4.%X11 := "DB_Drive_4UZ1".Status.%X4 AND ("DB_Drive_4UZ1".FaultCode = W#16#7788); // F30600
   "HMI_DB".Drives.Drive_4UZ1.Faults.FaultsWord4.%X12 := "DB_Drive_4UZ1".Status.%X4 AND ("DB_Drive_4UZ1".FaultCode = W#16#77C8); // F30664
   "HMI_DB".Drives.Drive_4UZ1.Faults.FaultsWord4.%X13 := "DB_Drive_4UZ1".Status.%X4 AND ("DB_Drive_4UZ1".FaultCode = W#16#7882); // F30850
   "HMI_DB".Drives.Drive_4UZ1.Faults.FaultsWord4.%X14 := "DB_Drive_4UZ1".Status.%X4 AND ("DB_Drive_4UZ1".FaultCode = W#16#1843); // F06211
   "HMI_DB".Drives.Drive_4UZ1.Faults.FaultsWord4.%X15 := "DB_Drive_4UZ1".Status.%X4 AND ("DB_Drive_4UZ1".FaultCode = W#16#213E); // F08510
END_REGION

REGION Network 5 (SCL): Формування слів аварій для HMI - ПЧ 4UZ2
   // ============================================================
   // 1. FaultsWord1
   // ============================================================

   "HMI_DB".Drives.Drive_4UZ2.Faults.FaultsWord1.%X0 := "DB_Drive_4UZ2".Status.%X4 AND ("DB_Drive_4UZ2".FaultCode = W#16#03E8); // F01000
   "HMI_DB".Drives.Drive_4UZ2.Faults.FaultsWord1.%X1 := "DB_Drive_4UZ2".Status.%X4 AND ("DB_Drive_4UZ2".FaultCode = W#16#03E9); // F01001
   "HMI_DB".Drives.Drive_4UZ2.Faults.FaultsWord1.%X2 := "DB_Drive_4UZ2".Status.%X4 AND ("DB_Drive_4UZ2".FaultCode = W#16#03F7); // F01015
   "HMI_DB".Drives.Drive_4UZ2.Faults.FaultsWord1.%X3 := "DB_Drive_4UZ2".Status.%X4 AND ("DB_Drive_4UZ2".FaultCode = W#16#0409); // F01033
   "HMI_DB".Drives.Drive_4UZ2.Faults.FaultsWord1.%X4 := "DB_Drive_4UZ2".Status.%X4 AND ("DB_Drive_4UZ2".FaultCode = W#16#040A); // F01034
   "HMI_DB".Drives.Drive_4UZ2.Faults.FaultsWord1.%X5 := "DB_Drive_4UZ2".Status.%X4 AND ("DB_Drive_4UZ2".FaultCode = W#16#0410); // F01040
   "HMI_DB".Drives.Drive_4UZ2.Faults.FaultsWord1.%X6 := "DB_Drive_4UZ2".Status.%X4 AND ("DB_Drive_4UZ2".FaultCode = W#16#0414); // F01044
   "HMI_DB".Drives.Drive_4UZ2.Faults.FaultsWord1.%X7 := "DB_Drive_4UZ2".Status.%X4 AND ("DB_Drive_4UZ2".FaultCode = W#16#041E); // F01054
   "HMI_DB".Drives.Drive_4UZ2.Faults.FaultsWord1.%X8 := "DB_Drive_4UZ2".Status.%X4 AND ("DB_Drive_4UZ2".FaultCode = W#16#0451); // F01105
   "HMI_DB".Drives.Drive_4UZ2.Faults.FaultsWord1.%X9 := "DB_Drive_4UZ2".Status.%X4 AND ("DB_Drive_4UZ2".FaultCode = W#16#0462); // F01122
   "HMI_DB".Drives.Drive_4UZ2.Faults.FaultsWord1.%X10 := "DB_Drive_4UZ2".Status.%X4 AND ("DB_Drive_4UZ2".FaultCode = W#16#04B5); // F01205
   "HMI_DB".Drives.Drive_4UZ2.Faults.FaultsWord1.%X11 := "DB_Drive_4UZ2".Status.%X4 AND ("DB_Drive_4UZ2".FaultCode = W#16#04E2); // F01250
   "HMI_DB".Drives.Drive_4UZ2.Faults.FaultsWord1.%X12 := "DB_Drive_4UZ2".Status.%X4 AND ("DB_Drive_4UZ2".FaultCode = W#16#05E8); // F01512
   "HMI_DB".Drives.Drive_4UZ2.Faults.FaultsWord1.%X13 := "DB_Drive_4UZ2".Status.%X4 AND ("DB_Drive_4UZ2".FaultCode = W#16#0640); // F01600
   "HMI_DB".Drives.Drive_4UZ2.Faults.FaultsWord1.%X14 := "DB_Drive_4UZ2".Status.%X4 AND ("DB_Drive_4UZ2".FaultCode = W#16#0659); // F01625
   "HMI_DB".Drives.Drive_4UZ2.Faults.FaultsWord1.%X15 := "DB_Drive_4UZ2".Status.%X4 AND ("DB_Drive_4UZ2".FaultCode = W#16#0672); // F01650


   // ============================================================
   // 2. FaultsWord2
   // ============================================================

   "HMI_DB".Drives.Drive_4UZ2.Faults.FaultsWord2.%X0 := "DB_Drive_4UZ2".Status.%X4 AND ("DB_Drive_4UZ2".FaultCode = W#16#067B); // F01659
   "HMI_DB".Drives.Drive_4UZ2.Faults.FaultsWord2.%X1 := "DB_Drive_4UZ2".Status.%X4 AND ("DB_Drive_4UZ2".FaultCode = W#16#0682); // F01666
   "HMI_DB".Drives.Drive_4UZ2.Faults.FaultsWord2.%X2 := "DB_Drive_4UZ2".Status.%X4 AND ("DB_Drive_4UZ2".FaultCode = W#16#0776); // F01910
   "HMI_DB".Drives.Drive_4UZ2.Faults.FaultsWord2.%X3 := "DB_Drive_4UZ2".Status.%X4 AND ("DB_Drive_4UZ2".FaultCode = W#16#18A6); // F06310
   "HMI_DB".Drives.Drive_4UZ2.Faults.FaultsWord2.%X4 := "DB_Drive_4UZ2".Status.%X4 AND ("DB_Drive_4UZ2".FaultCode = W#16#1B63); // F07011
   "HMI_DB".Drives.Drive_4UZ2.Faults.FaultsWord2.%X5 := "DB_Drive_4UZ2".Status.%X4 AND ("DB_Drive_4UZ2".FaultCode = W#16#1B68); // F07016
   "HMI_DB".Drives.Drive_4UZ2.Faults.FaultsWord2.%X6 := "DB_Drive_4UZ2".Status.%X4 AND ("DB_Drive_4UZ2".FaultCode = W#16#1BAE); // F07086
   "HMI_DB".Drives.Drive_4UZ2.Faults.FaultsWord2.%X7 := "DB_Drive_4UZ2".Status.%X4 AND ("DB_Drive_4UZ2".FaultCode = W#16#1BB0); // F07088
   "HMI_DB".Drives.Drive_4UZ2.Faults.FaultsWord2.%X8 := "DB_Drive_4UZ2".Status.%X4 AND ("DB_Drive_4UZ2".FaultCode = W#16#1C98); // F07320
   "HMI_DB".Drives.Drive_4UZ2.Faults.FaultsWord2.%X9 := "DB_Drive_4UZ2".Status.%X4 AND ("DB_Drive_4UZ2".FaultCode = W#16#1CA2); // F07330
   "HMI_DB".Drives.Drive_4UZ2.Faults.FaultsWord2.%X10 := "DB_Drive_4UZ2".Status.%X4 AND ("DB_Drive_4UZ2".FaultCode = W#16#1D02); // F07426
   "HMI_DB".Drives.Drive_4UZ2.Faults.FaultsWord2.%X11 := "DB_Drive_4UZ2".Status.%X4 AND ("DB_Drive_4UZ2".FaultCode = W#16#1E79); // F07801
   "HMI_DB".Drives.Drive_4UZ2.Faults.FaultsWord2.%X12 := "DB_Drive_4UZ2".Status.%X4 AND ("DB_Drive_4UZ2".FaultCode = W#16#1E7F); // F07807
   "HMI_DB".Drives.Drive_4UZ2.Faults.FaultsWord2.%X13 := "DB_Drive_4UZ2".Status.%X4 AND ("DB_Drive_4UZ2".FaultCode = W#16#1EB4); // F07860
   "HMI_DB".Drives.Drive_4UZ2.Faults.FaultsWord2.%X14 := "DB_Drive_4UZ2".Status.%X4 AND ("DB_Drive_4UZ2".FaultCode = W#16#1EB5); // F07861
   "HMI_DB".Drives.Drive_4UZ2.Faults.FaultsWord2.%X15 := "DB_Drive_4UZ2".Status.%X4 AND ("DB_Drive_4UZ2".FaultCode = W#16#1EB6); // F07862


   // ============================================================
   // 3. FaultsWord3
   // ============================================================

   "HMI_DB".Drives.Drive_4UZ2.Faults.FaultsWord3.%X0 := "DB_Drive_4UZ2".Status.%X4 AND ("DB_Drive_4UZ2".FaultCode = W#16#1EDC); // F07900
   "HMI_DB".Drives.Drive_4UZ2.Faults.FaultsWord3.%X1 := "DB_Drive_4UZ2".Status.%X4 AND ("DB_Drive_4UZ2".FaultCode = W#16#1EDD); // F07901
   "HMI_DB".Drives.Drive_4UZ2.Faults.FaultsWord3.%X2 := "DB_Drive_4UZ2".Status.%X4 AND ("DB_Drive_4UZ2".FaultCode = W#16#1EDE); // F07902
   "HMI_DB".Drives.Drive_4UZ2.Faults.FaultsWord3.%X3 := "DB_Drive_4UZ2".Status.%X4 AND ("DB_Drive_4UZ2".FaultCode = W#16#1EF3); // F07923
   "HMI_DB".Drives.Drive_4UZ2.Faults.FaultsWord3.%X4 := "DB_Drive_4UZ2".Status.%X4 AND ("DB_Drive_4UZ2".FaultCode = W#16#1EF4); // F07924
   "HMI_DB".Drives.Drive_4UZ2.Faults.FaultsWord3.%X5 := "DB_Drive_4UZ2".Status.%X4 AND ("DB_Drive_4UZ2".FaultCode = W#16#2135); // F08501
   "HMI_DB".Drives.Drive_4UZ2.Faults.FaultsWord3.%X6 := "DB_Drive_4UZ2".Status.%X4 AND ("DB_Drive_4UZ2".FaultCode = W#16#2136); // F08502
   "HMI_DB".Drives.Drive_4UZ2.Faults.FaultsWord3.%X7 := "DB_Drive_4UZ2".Status.%X4 AND ("DB_Drive_4UZ2".FaultCode = W#16#1842); // F06210
   "HMI_DB".Drives.Drive_4UZ2.Faults.FaultsWord3.%X8 := "DB_Drive_4UZ2".Status.%X4 AND ("DB_Drive_4UZ2".FaultCode = W#16#332C); // F13100
   "HMI_DB".Drives.Drive_4UZ2.Faults.FaultsWord3.%X9 := "DB_Drive_4UZ2".Status.%X4 AND ("DB_Drive_4UZ2".FaultCode = W#16#332D); // F13101
   "HMI_DB".Drives.Drive_4UZ2.Faults.FaultsWord3.%X10 := "DB_Drive_4UZ2".Status.%X4 AND ("DB_Drive_4UZ2".FaultCode = W#16#7531); // F30001
   "HMI_DB".Drives.Drive_4UZ2.Faults.FaultsWord3.%X11 := "DB_Drive_4UZ2".Status.%X4 AND ("DB_Drive_4UZ2".FaultCode = W#16#7532); // F30002
   "HMI_DB".Drives.Drive_4UZ2.Faults.FaultsWord3.%X12 := "DB_Drive_4UZ2".Status.%X4 AND ("DB_Drive_4UZ2".FaultCode = W#16#7533); // F30003
   "HMI_DB".Drives.Drive_4UZ2.Faults.FaultsWord3.%X13 := "DB_Drive_4UZ2".Status.%X4 AND ("DB_Drive_4UZ2".FaultCode = W#16#7534); // F30004
   "HMI_DB".Drives.Drive_4UZ2.Faults.FaultsWord3.%X14 := "DB_Drive_4UZ2".Status.%X4 AND ("DB_Drive_4UZ2".FaultCode = W#16#7535); // F30005
   "HMI_DB".Drives.Drive_4UZ2.Faults.FaultsWord3.%X15 := "DB_Drive_4UZ2".Status.%X4 AND ("DB_Drive_4UZ2".FaultCode = W#16#753B); // F30011


   // ============================================================
   // 4. FaultsWord4
   // ============================================================

   "HMI_DB".Drives.Drive_4UZ2.Faults.FaultsWord4.%X0 := "DB_Drive_4UZ2".Status.%X4 AND ("DB_Drive_4UZ2".FaultCode = W#16#753F); // F30015
   "HMI_DB".Drives.Drive_4UZ2.Faults.FaultsWord4.%X1 := "DB_Drive_4UZ2".Status.%X4 AND ("DB_Drive_4UZ2".FaultCode = W#16#7545); // F30021
   "HMI_DB".Drives.Drive_4UZ2.Faults.FaultsWord4.%X2 := "DB_Drive_4UZ2".Status.%X4 AND ("DB_Drive_4UZ2".FaultCode = W#16#7546); // F30022
   "HMI_DB".Drives.Drive_4UZ2.Faults.FaultsWord4.%X3 := "DB_Drive_4UZ2".Status.%X4 AND ("DB_Drive_4UZ2".FaultCode = W#16#754B); // F30027
   "HMI_DB".Drives.Drive_4UZ2.Faults.FaultsWord4.%X4 := "DB_Drive_4UZ2".Status.%X4 AND ("DB_Drive_4UZ2".FaultCode = W#16#7553); // F30035
   "HMI_DB".Drives.Drive_4UZ2.Faults.FaultsWord4.%X5 := "DB_Drive_4UZ2".Status.%X4 AND ("DB_Drive_4UZ2".FaultCode = W#16#7554); // F30036
   "HMI_DB".Drives.Drive_4UZ2.Faults.FaultsWord4.%X6 := "DB_Drive_4UZ2".Status.%X4 AND ("DB_Drive_4UZ2".FaultCode = W#16#7555); // F30037
   "HMI_DB".Drives.Drive_4UZ2.Faults.FaultsWord4.%X7 := "DB_Drive_4UZ2".Status.%X4 AND ("DB_Drive_4UZ2".FaultCode = W#16#7564); // F30052
   "HMI_DB".Drives.Drive_4UZ2.Faults.FaultsWord4.%X8 := "DB_Drive_4UZ2".Status.%X4 AND ("DB_Drive_4UZ2".FaultCode = W#16#7565); // F30053
   "HMI_DB".Drives.Drive_4UZ2.Faults.FaultsWord4.%X9 := "DB_Drive_4UZ2".Status.%X4 AND ("DB_Drive_4UZ2".FaultCode = W#16#756B); // F30059
   "HMI_DB".Drives.Drive_4UZ2.Faults.FaultsWord4.%X10 := "DB_Drive_4UZ2".Status.%X4 AND ("DB_Drive_4UZ2".FaultCode = W#16#757A); // F30074
   "HMI_DB".Drives.Drive_4UZ2.Faults.FaultsWord4.%X11 := "DB_Drive_4UZ2".Status.%X4 AND ("DB_Drive_4UZ2".FaultCode = W#16#7788); // F30600
   "HMI_DB".Drives.Drive_4UZ2.Faults.FaultsWord4.%X12 := "DB_Drive_4UZ2".Status.%X4 AND ("DB_Drive_4UZ2".FaultCode = W#16#77C8); // F30664
   "HMI_DB".Drives.Drive_4UZ2.Faults.FaultsWord4.%X13 := "DB_Drive_4UZ2".Status.%X4 AND ("DB_Drive_4UZ2".FaultCode = W#16#7882); // F30850
   "HMI_DB".Drives.Drive_4UZ2.Faults.FaultsWord4.%X14 := "DB_Drive_4UZ2".Status.%X4 AND ("DB_Drive_4UZ2".FaultCode = W#16#1843); // F06211
   "HMI_DB".Drives.Drive_4UZ2.Faults.FaultsWord4.%X15 := "DB_Drive_4UZ2".Status.%X4 AND ("DB_Drive_4UZ2".FaultCode = W#16#213E); // F08510
END_REGION
END_FUNCTION

FUNCTION "FC_Drives_HMI_Warnings" : Void   // FC54, LAD
TITLE = Формування слів попереджень (Alarms) ПЧ для HMI
{ S7_Optimized_Access := 'TRUE' }
VERSION : 0.1
BEGIN

REGION Network 2 (SCL): Формування слів попереджень для HMI - ПЧ 1UZ1
   // ============================================================
   // 1. AlarmsWord1
   // ============================================================

   "HMI_DB".Drives.Drive_1UZ1.Alarms.AlarmsWord1.%X0 := "DB_Drive_1UZ1".Status.%X5 AND ("DB_Drive_1UZ1".WarningCode = W#16#0636); // A01590
   "HMI_DB".Drives.Drive_1UZ1.Alarms.AlarmsWord1.%X1 := "DB_Drive_1UZ1".Status.%X5 AND ("DB_Drive_1UZ1".WarningCode = W#16#0682); // A01666
   "HMI_DB".Drives.Drive_1UZ1.Alarms.AlarmsWord1.%X2 := "DB_Drive_1UZ1".Status.%X5 AND ("DB_Drive_1UZ1".WarningCode = W#16#06A2); // A01698
   "HMI_DB".Drives.Drive_1UZ1.Alarms.AlarmsWord1.%X3 := "DB_Drive_1UZ1".Status.%X5 AND ("DB_Drive_1UZ1".WarningCode = W#16#06A3); // A01699
   "HMI_DB".Drives.Drive_1UZ1.Alarms.AlarmsWord1.%X4 := "DB_Drive_1UZ1".Status.%X5 AND ("DB_Drive_1UZ1".WarningCode = W#16#076C); // A01900
   "HMI_DB".Drives.Drive_1UZ1.Alarms.AlarmsWord1.%X5 := "DB_Drive_1UZ1".Status.%X5 AND ("DB_Drive_1UZ1".WarningCode = W#16#0780); // A01920
   "HMI_DB".Drives.Drive_1UZ1.Alarms.AlarmsWord1.%X6 := "DB_Drive_1UZ1".Status.%X5 AND ("DB_Drive_1UZ1".WarningCode = W#16#1388); // A05000
   "HMI_DB".Drives.Drive_1UZ1.Alarms.AlarmsWord1.%X7 := "DB_Drive_1UZ1".Status.%X5 AND ("DB_Drive_1UZ1".WarningCode = W#16#1389); // A05001
   "HMI_DB".Drives.Drive_1UZ1.Alarms.AlarmsWord1.%X8 := "DB_Drive_1UZ1".Status.%X5 AND ("DB_Drive_1UZ1".WarningCode = W#16#138A); // A05002
   "HMI_DB".Drives.Drive_1UZ1.Alarms.AlarmsWord1.%X9 := "DB_Drive_1UZ1".Status.%X5 AND ("DB_Drive_1UZ1".WarningCode = W#16#138C); // A05004
   "HMI_DB".Drives.Drive_1UZ1.Alarms.AlarmsWord1.%X10 := "DB_Drive_1UZ1".Status.%X5 AND ("DB_Drive_1UZ1".WarningCode = W#16#138E); // A05006
   "HMI_DB".Drives.Drive_1UZ1.Alarms.AlarmsWord1.%X11 := "DB_Drive_1UZ1".Status.%X5 AND ("DB_Drive_1UZ1".WarningCode = W#16#1B64); // A07012
   "HMI_DB".Drives.Drive_1UZ1.Alarms.AlarmsWord1.%X12 := "DB_Drive_1UZ1".Status.%X5 AND ("DB_Drive_1UZ1".WarningCode = W#16#03F5); // A01013
   "HMI_DB".Drives.Drive_1UZ1.Alarms.AlarmsWord1.%X13 := "DB_Drive_1UZ1".Status.%X5 AND ("DB_Drive_1UZ1".WarningCode = W#16#1C99); // A07321
   "HMI_DB".Drives.Drive_1UZ1.Alarms.AlarmsWord1.%X14 := "DB_Drive_1UZ1".Status.%X5 AND ("DB_Drive_1UZ1".WarningCode = W#16#1CE8); // A07400
   "HMI_DB".Drives.Drive_1UZ1.Alarms.AlarmsWord1.%X15 := "DB_Drive_1UZ1".Status.%X5 AND ("DB_Drive_1UZ1".WarningCode = W#16#1CF1); // A07409

   // ============================================================
   // 2. AlarmsWord2
   // ============================================================

   "HMI_DB".Drives.Drive_1UZ1.Alarms.AlarmsWord2.%X0 := "DB_Drive_1UZ1".Status.%X5 AND ("DB_Drive_1UZ1".WarningCode = W#16#1E7D); // A07805
   "HMI_DB".Drives.Drive_1UZ1.Alarms.AlarmsWord2.%X1 := "DB_Drive_1UZ1".Status.%X5 AND ("DB_Drive_1UZ1".WarningCode = W#16#1EAA); // A07850
   "HMI_DB".Drives.Drive_1UZ1.Alarms.AlarmsWord2.%X2 := "DB_Drive_1UZ1".Status.%X5 AND ("DB_Drive_1UZ1".WarningCode = W#16#1EAB); // A07851
   "HMI_DB".Drives.Drive_1UZ1.Alarms.AlarmsWord2.%X3 := "DB_Drive_1UZ1".Status.%X5 AND ("DB_Drive_1UZ1".WarningCode = W#16#1EAC); // A07852
   "HMI_DB".Drives.Drive_1UZ1.Alarms.AlarmsWord2.%X4 := "DB_Drive_1UZ1".Status.%X5 AND ("DB_Drive_1UZ1".WarningCode = W#16#1EDF); // A07903
   "HMI_DB".Drives.Drive_1UZ1.Alarms.AlarmsWord2.%X5 := "DB_Drive_1UZ1".Status.%X5 AND ("DB_Drive_1UZ1".WarningCode = W#16#1EE6); // A07910
   "HMI_DB".Drives.Drive_1UZ1.Alarms.AlarmsWord2.%X6 := "DB_Drive_1UZ1".Status.%X5 AND ("DB_Drive_1UZ1".WarningCode = W#16#1EF0); // A07920
   "HMI_DB".Drives.Drive_1UZ1.Alarms.AlarmsWord2.%X7 := "DB_Drive_1UZ1".Status.%X5 AND ("DB_Drive_1UZ1".WarningCode = W#16#1EF1); // A07921
   "HMI_DB".Drives.Drive_1UZ1.Alarms.AlarmsWord2.%X8 := "DB_Drive_1UZ1".Status.%X5 AND ("DB_Drive_1UZ1".WarningCode = W#16#1EF2); // A07922
   "HMI_DB".Drives.Drive_1UZ1.Alarms.AlarmsWord2.%X9 := "DB_Drive_1UZ1".Status.%X5 AND ("DB_Drive_1UZ1".WarningCode = W#16#1EF7); // A07927
   "HMI_DB".Drives.Drive_1UZ1.Alarms.AlarmsWord2.%X10 := "DB_Drive_1UZ1".Status.%X5 AND ("DB_Drive_1UZ1".WarningCode = W#16#1F2C); // A07980
   "HMI_DB".Drives.Drive_1UZ1.Alarms.AlarmsWord2.%X11 := "DB_Drive_1UZ1".Status.%X5 AND ("DB_Drive_1UZ1".WarningCode = W#16#1F2D); // A07981
   "HMI_DB".Drives.Drive_1UZ1.Alarms.AlarmsWord2.%X12 := "DB_Drive_1UZ1".Status.%X5 AND ("DB_Drive_1UZ1".WarningCode = W#16#1F37); // A07991
   "HMI_DB".Drives.Drive_1UZ1.Alarms.AlarmsWord2.%X13 := "DB_Drive_1UZ1".Status.%X5 AND ("DB_Drive_1UZ1".WarningCode = W#16#213F); // A08511
   "HMI_DB".Drives.Drive_1UZ1.Alarms.AlarmsWord2.%X14 := "DB_Drive_1UZ1".Status.%X5 AND ("DB_Drive_1UZ1".WarningCode = W#16#214E); // A08526
   "HMI_DB".Drives.Drive_1UZ1.Alarms.AlarmsWord2.%X15 := "DB_Drive_1UZ1".Status.%X5 AND ("DB_Drive_1UZ1".WarningCode = W#16#2175); // A08565


   // ============================================================
   // 3. AlarmsWord3
   // ============================================================

   "HMI_DB".Drives.Drive_1UZ1.Alarms.AlarmsWord3.%X0 := "DB_Drive_1UZ1".Status.%X5 AND ("DB_Drive_1UZ1".WarningCode = W#16#7561); // A30049
   "HMI_DB".Drives.Drive_1UZ1.Alarms.AlarmsWord3.%X1 := "DB_Drive_1UZ1".Status.%X5 AND ("DB_Drive_1UZ1".WarningCode = W#16#7726); // A30502
   "HMI_DB".Drives.Drive_1UZ1.Alarms.AlarmsWord3.%X2 := "DB_Drive_1UZ1".Status.%X5 AND ("DB_Drive_1UZ1".WarningCode = W#16#78C8); // A30920
   "HMI_DB".Drives.Drive_1UZ1.Alarms.AlarmsWord3.%X3 := "DB_Drive_1UZ1".Status.%X5 AND ("DB_Drive_1UZ1".WarningCode = W#16#183D); // A06205
   "HMI_DB".Drives.Drive_1UZ1.Alarms.AlarmsWord3.%X4 := "DB_Drive_1UZ1".Status.%X5 AND ("DB_Drive_1UZ1".WarningCode = W#16#183E); // A06206
   "HMI_DB".Drives.Drive_1UZ1.Alarms.AlarmsWord3.%X5 := "DB_Drive_1UZ1".Status.%X5 AND ("DB_Drive_1UZ1".WarningCode = W#16#1840); // A06208
   "HMI_DB".Drives.Drive_1UZ1.Alarms.AlarmsWord3.%X6 := "DB_Drive_1UZ1".Status.%X5 AND ("DB_Drive_1UZ1".WarningCode = W#16#1847); // A06215
   "HMI_DB".Drives.Drive_1UZ1.Alarms.AlarmsWord3.%X7 := "DB_Drive_1UZ1".Status.%X5 AND ("DB_Drive_1UZ1".WarningCode = W#16#186A); // A06250
   "HMI_DB".Drives.Drive_1UZ1.Alarms.AlarmsWord3.%X8 := "DB_Drive_1UZ1".Status.%X5 AND ("DB_Drive_1UZ1".WarningCode = W#16#1874); // A06260
   "HMI_DB".Drives.Drive_1UZ1.Alarms.AlarmsWord3.%X9 := "DB_Drive_1UZ1".Status.%X5 AND ("DB_Drive_1UZ1".WarningCode = W#16#189D); // A06301
   "HMI_DB".Drives.Drive_1UZ1.Alarms.AlarmsWord3.%X10 := "DB_Drive_1UZ1".Status.%X5 AND ("DB_Drive_1UZ1".WarningCode = W#16#18CE); // A06350
   "HMI_DB".Drives.Drive_1UZ1.Alarms.AlarmsWord3.%X11 := "DB_Drive_1UZ1".Status.%X5 AND ("DB_Drive_1UZ1".WarningCode = W#16#18CF); // A06351
   "HMI_DB".Drives.Drive_1UZ1.Alarms.AlarmsWord3.%X12 := "DB_Drive_1UZ1".Status.%X5 AND ("DB_Drive_1UZ1".WarningCode = W#16#1A90); // A06800
   "HMI_DB".Drives.Drive_1UZ1.Alarms.AlarmsWord3.%X13 := "DB_Drive_1UZ1".Status.%X5 AND ("DB_Drive_1UZ1".WarningCode = W#16#7552); // A30034
   "HMI_DB".Drives.Drive_1UZ1.Alarms.AlarmsWord3.%X14 := "DB_Drive_1UZ1".Status.%X5 AND ("DB_Drive_1UZ1".WarningCode = W#16#7559); // A30041
   "HMI_DB".Drives.Drive_1UZ1.Alarms.AlarmsWord3.%X15 := "DB_Drive_1UZ1".Status.%X5 AND ("DB_Drive_1UZ1".WarningCode = W#16#755A); // A30042


   // ============================================================
   // 4. AlarmsWord4
   // ============================================================

   "HMI_DB".Drives.Drive_1UZ1.Alarms.AlarmsWord4.%X0 := "DB_Drive_1UZ1".Status.%X5 AND ("DB_Drive_1UZ1".WarningCode = W#16#755C); // A30044
   "HMI_DB".Drives.Drive_1UZ1.Alarms.AlarmsWord4.%X1 := "DB_Drive_1UZ1".Status.%X5 AND ("DB_Drive_1UZ1".WarningCode = W#16#755E); // A30046
   "HMI_DB".Drives.Drive_1UZ1.Alarms.AlarmsWord4.%X2 := "DB_Drive_1UZ1".Status.%X5 AND ("DB_Drive_1UZ1".WarningCode = W#16#757D); // A30077
   "HMI_DB".Drives.Drive_1UZ1.Alarms.AlarmsWord4.%X3 := "DB_Drive_1UZ1".Status.%X5 AND ("DB_Drive_1UZ1".WarningCode = W#16#757F); // A30079

   // Невикористані біти
   "HMI_DB".Drives.Drive_1UZ1.Alarms.AlarmsWord4.%X4 := FALSE;
   "HMI_DB".Drives.Drive_1UZ1.Alarms.AlarmsWord4.%X5 := FALSE;
   "HMI_DB".Drives.Drive_1UZ1.Alarms.AlarmsWord4.%X6 := FALSE;
   "HMI_DB".Drives.Drive_1UZ1.Alarms.AlarmsWord4.%X7 := FALSE;
   "HMI_DB".Drives.Drive_1UZ1.Alarms.AlarmsWord4.%X8 := FALSE;
   "HMI_DB".Drives.Drive_1UZ1.Alarms.AlarmsWord4.%X9 := FALSE;
   "HMI_DB".Drives.Drive_1UZ1.Alarms.AlarmsWord4.%X10 := FALSE;
   "HMI_DB".Drives.Drive_1UZ1.Alarms.AlarmsWord4.%X11 := FALSE;
   "HMI_DB".Drives.Drive_1UZ1.Alarms.AlarmsWord4.%X12 := FALSE;
   "HMI_DB".Drives.Drive_1UZ1.Alarms.AlarmsWord4.%X13 := FALSE;
   "HMI_DB".Drives.Drive_1UZ1.Alarms.AlarmsWord4.%X14 := FALSE;
   "HMI_DB".Drives.Drive_1UZ1.Alarms.AlarmsWord4.%X15 := FALSE;
END_REGION

REGION Network 3 (SCL): Формування слів попереджень для HMI - ПЧ 3UZ1
   // ============================================================
   // 1. AlarmsWord1
   // ============================================================

   "HMI_DB".Drives.Drive_3UZ1.Alarms.AlarmsWord1.%X0 := "DB_Drive_3UZ1".Status.%X5 AND ("DB_Drive_3UZ1".WarningCode = W#16#0636); // A01590
   "HMI_DB".Drives.Drive_3UZ1.Alarms.AlarmsWord1.%X1 := "DB_Drive_3UZ1".Status.%X5 AND ("DB_Drive_3UZ1".WarningCode = W#16#0682); // A01666
   "HMI_DB".Drives.Drive_3UZ1.Alarms.AlarmsWord1.%X2 := "DB_Drive_3UZ1".Status.%X5 AND ("DB_Drive_3UZ1".WarningCode = W#16#06A2); // A01698
   "HMI_DB".Drives.Drive_3UZ1.Alarms.AlarmsWord1.%X3 := "DB_Drive_3UZ1".Status.%X5 AND ("DB_Drive_3UZ1".WarningCode = W#16#06A3); // A01699
   "HMI_DB".Drives.Drive_3UZ1.Alarms.AlarmsWord1.%X4 := "DB_Drive_3UZ1".Status.%X5 AND ("DB_Drive_3UZ1".WarningCode = W#16#076C); // A01900
   "HMI_DB".Drives.Drive_3UZ1.Alarms.AlarmsWord1.%X5 := "DB_Drive_3UZ1".Status.%X5 AND ("DB_Drive_3UZ1".WarningCode = W#16#0780); // A01920
   "HMI_DB".Drives.Drive_3UZ1.Alarms.AlarmsWord1.%X6 := "DB_Drive_3UZ1".Status.%X5 AND ("DB_Drive_3UZ1".WarningCode = W#16#1388); // A05000
   "HMI_DB".Drives.Drive_3UZ1.Alarms.AlarmsWord1.%X7 := "DB_Drive_3UZ1".Status.%X5 AND ("DB_Drive_3UZ1".WarningCode = W#16#1389); // A05001
   "HMI_DB".Drives.Drive_3UZ1.Alarms.AlarmsWord1.%X8 := "DB_Drive_3UZ1".Status.%X5 AND ("DB_Drive_3UZ1".WarningCode = W#16#138A); // A05002
   "HMI_DB".Drives.Drive_3UZ1.Alarms.AlarmsWord1.%X9 := "DB_Drive_3UZ1".Status.%X5 AND ("DB_Drive_3UZ1".WarningCode = W#16#138C); // A05004
   "HMI_DB".Drives.Drive_3UZ1.Alarms.AlarmsWord1.%X10 := "DB_Drive_3UZ1".Status.%X5 AND ("DB_Drive_3UZ1".WarningCode = W#16#138E); // A05006
   "HMI_DB".Drives.Drive_3UZ1.Alarms.AlarmsWord1.%X11 := "DB_Drive_3UZ1".Status.%X5 AND ("DB_Drive_3UZ1".WarningCode = W#16#1B64); // A07012
   "HMI_DB".Drives.Drive_3UZ1.Alarms.AlarmsWord1.%X12 := "DB_Drive_3UZ1".Status.%X5 AND ("DB_Drive_3UZ1".WarningCode = W#16#03F5); // A01013
   "HMI_DB".Drives.Drive_3UZ1.Alarms.AlarmsWord1.%X13 := "DB_Drive_3UZ1".Status.%X5 AND ("DB_Drive_3UZ1".WarningCode = W#16#1C99); // A07321
   "HMI_DB".Drives.Drive_3UZ1.Alarms.AlarmsWord1.%X14 := "DB_Drive_3UZ1".Status.%X5 AND ("DB_Drive_3UZ1".WarningCode = W#16#1CE8); // A07400
   "HMI_DB".Drives.Drive_3UZ1.Alarms.AlarmsWord1.%X15 := "DB_Drive_3UZ1".Status.%X5 AND ("DB_Drive_3UZ1".WarningCode = W#16#1CF1); // A07409

   // ============================================================
   // 2. AlarmsWord2
   // ============================================================

   "HMI_DB".Drives.Drive_3UZ1.Alarms.AlarmsWord2.%X0 := "DB_Drive_3UZ1".Status.%X5 AND ("DB_Drive_3UZ1".WarningCode = W#16#1E7D); // A07805
   "HMI_DB".Drives.Drive_3UZ1.Alarms.AlarmsWord2.%X1 := "DB_Drive_3UZ1".Status.%X5 AND ("DB_Drive_3UZ1".WarningCode = W#16#1EAA); // A07850
   "HMI_DB".Drives.Drive_3UZ1.Alarms.AlarmsWord2.%X2 := "DB_Drive_3UZ1".Status.%X5 AND ("DB_Drive_3UZ1".WarningCode = W#16#1EAB); // A07851
   "HMI_DB".Drives.Drive_3UZ1.Alarms.AlarmsWord2.%X3 := "DB_Drive_3UZ1".Status.%X5 AND ("DB_Drive_3UZ1".WarningCode = W#16#1EAC); // A07852
   "HMI_DB".Drives.Drive_3UZ1.Alarms.AlarmsWord2.%X4 := "DB_Drive_3UZ1".Status.%X5 AND ("DB_Drive_3UZ1".WarningCode = W#16#1EDF); // A07903
   "HMI_DB".Drives.Drive_3UZ1.Alarms.AlarmsWord2.%X5 := "DB_Drive_3UZ1".Status.%X5 AND ("DB_Drive_3UZ1".WarningCode = W#16#1EE6); // A07910
   "HMI_DB".Drives.Drive_3UZ1.Alarms.AlarmsWord2.%X6 := "DB_Drive_3UZ1".Status.%X5 AND ("DB_Drive_3UZ1".WarningCode = W#16#1EF0); // A07920
   "HMI_DB".Drives.Drive_3UZ1.Alarms.AlarmsWord2.%X7 := "DB_Drive_3UZ1".Status.%X5 AND ("DB_Drive_3UZ1".WarningCode = W#16#1EF1); // A07921
   "HMI_DB".Drives.Drive_3UZ1.Alarms.AlarmsWord2.%X8 := "DB_Drive_3UZ1".Status.%X5 AND ("DB_Drive_3UZ1".WarningCode = W#16#1EF2); // A07922
   "HMI_DB".Drives.Drive_3UZ1.Alarms.AlarmsWord2.%X9 := "DB_Drive_3UZ1".Status.%X5 AND ("DB_Drive_3UZ1".WarningCode = W#16#1EF7); // A07927
   "HMI_DB".Drives.Drive_3UZ1.Alarms.AlarmsWord2.%X10 := "DB_Drive_3UZ1".Status.%X5 AND ("DB_Drive_3UZ1".WarningCode = W#16#1F2C); // A07980
   "HMI_DB".Drives.Drive_3UZ1.Alarms.AlarmsWord2.%X11 := "DB_Drive_3UZ1".Status.%X5 AND ("DB_Drive_3UZ1".WarningCode = W#16#1F2D); // A07981
   "HMI_DB".Drives.Drive_3UZ1.Alarms.AlarmsWord2.%X12 := "DB_Drive_3UZ1".Status.%X5 AND ("DB_Drive_3UZ1".WarningCode = W#16#1F37); // A07991
   "HMI_DB".Drives.Drive_3UZ1.Alarms.AlarmsWord2.%X13 := "DB_Drive_3UZ1".Status.%X5 AND ("DB_Drive_3UZ1".WarningCode = W#16#213F); // A08511
   "HMI_DB".Drives.Drive_3UZ1.Alarms.AlarmsWord2.%X14 := "DB_Drive_3UZ1".Status.%X5 AND ("DB_Drive_3UZ1".WarningCode = W#16#214E); // A08526
   "HMI_DB".Drives.Drive_3UZ1.Alarms.AlarmsWord2.%X15 := "DB_Drive_3UZ1".Status.%X5 AND ("DB_Drive_3UZ1".WarningCode = W#16#2175); // A08565


   // ============================================================
   // 3. AlarmsWord3
   // ============================================================

   "HMI_DB".Drives.Drive_3UZ1.Alarms.AlarmsWord3.%X0 := "DB_Drive_3UZ1".Status.%X5 AND ("DB_Drive_3UZ1".WarningCode = W#16#7561); // A30049
   "HMI_DB".Drives.Drive_3UZ1.Alarms.AlarmsWord3.%X1 := "DB_Drive_3UZ1".Status.%X5 AND ("DB_Drive_3UZ1".WarningCode = W#16#7726); // A30502
   "HMI_DB".Drives.Drive_3UZ1.Alarms.AlarmsWord3.%X2 := "DB_Drive_3UZ1".Status.%X5 AND ("DB_Drive_3UZ1".WarningCode = W#16#78C8); // A30920
   "HMI_DB".Drives.Drive_3UZ1.Alarms.AlarmsWord3.%X3 := "DB_Drive_3UZ1".Status.%X5 AND ("DB_Drive_3UZ1".WarningCode = W#16#183D); // A06205
   "HMI_DB".Drives.Drive_3UZ1.Alarms.AlarmsWord3.%X4 := "DB_Drive_3UZ1".Status.%X5 AND ("DB_Drive_3UZ1".WarningCode = W#16#183E); // A06206
   "HMI_DB".Drives.Drive_3UZ1.Alarms.AlarmsWord3.%X5 := "DB_Drive_3UZ1".Status.%X5 AND ("DB_Drive_3UZ1".WarningCode = W#16#1840); // A06208
   "HMI_DB".Drives.Drive_3UZ1.Alarms.AlarmsWord3.%X6 := "DB_Drive_3UZ1".Status.%X5 AND ("DB_Drive_3UZ1".WarningCode = W#16#1847); // A06215
   "HMI_DB".Drives.Drive_3UZ1.Alarms.AlarmsWord3.%X7 := "DB_Drive_3UZ1".Status.%X5 AND ("DB_Drive_3UZ1".WarningCode = W#16#186A); // A06250
   "HMI_DB".Drives.Drive_3UZ1.Alarms.AlarmsWord3.%X8 := "DB_Drive_3UZ1".Status.%X5 AND ("DB_Drive_3UZ1".WarningCode = W#16#1874); // A06260
   "HMI_DB".Drives.Drive_3UZ1.Alarms.AlarmsWord3.%X9 := "DB_Drive_3UZ1".Status.%X5 AND ("DB_Drive_3UZ1".WarningCode = W#16#189D); // A06301
   "HMI_DB".Drives.Drive_3UZ1.Alarms.AlarmsWord3.%X10 := "DB_Drive_3UZ1".Status.%X5 AND ("DB_Drive_3UZ1".WarningCode = W#16#18CE); // A06350
   "HMI_DB".Drives.Drive_3UZ1.Alarms.AlarmsWord3.%X11 := "DB_Drive_3UZ1".Status.%X5 AND ("DB_Drive_3UZ1".WarningCode = W#16#18CF); // A06351
   "HMI_DB".Drives.Drive_3UZ1.Alarms.AlarmsWord3.%X12 := "DB_Drive_3UZ1".Status.%X5 AND ("DB_Drive_3UZ1".WarningCode = W#16#1A90); // A06800
   "HMI_DB".Drives.Drive_3UZ1.Alarms.AlarmsWord3.%X13 := "DB_Drive_3UZ1".Status.%X5 AND ("DB_Drive_3UZ1".WarningCode = W#16#7552); // A30034
   "HMI_DB".Drives.Drive_3UZ1.Alarms.AlarmsWord3.%X14 := "DB_Drive_3UZ1".Status.%X5 AND ("DB_Drive_3UZ1".WarningCode = W#16#7559); // A30041
   "HMI_DB".Drives.Drive_3UZ1.Alarms.AlarmsWord3.%X15 := "DB_Drive_3UZ1".Status.%X5 AND ("DB_Drive_3UZ1".WarningCode = W#16#755A); // A30042


   // ============================================================
   // 4. AlarmsWord4
   // ============================================================

   "HMI_DB".Drives.Drive_3UZ1.Alarms.AlarmsWord4.%X0 := "DB_Drive_3UZ1".Status.%X5 AND ("DB_Drive_3UZ1".WarningCode = W#16#755C); // A30044
   "HMI_DB".Drives.Drive_3UZ1.Alarms.AlarmsWord4.%X1 := "DB_Drive_3UZ1".Status.%X5 AND ("DB_Drive_3UZ1".WarningCode = W#16#755E); // A30046
   "HMI_DB".Drives.Drive_3UZ1.Alarms.AlarmsWord4.%X2 := "DB_Drive_3UZ1".Status.%X5 AND ("DB_Drive_3UZ1".WarningCode = W#16#757D); // A30077
   "HMI_DB".Drives.Drive_3UZ1.Alarms.AlarmsWord4.%X3 := "DB_Drive_3UZ1".Status.%X5 AND ("DB_Drive_3UZ1".WarningCode = W#16#757F); // A30079

   // Невикористані біти
   "HMI_DB".Drives.Drive_3UZ1.Alarms.AlarmsWord4.%X4 := FALSE;
   "HMI_DB".Drives.Drive_3UZ1.Alarms.AlarmsWord4.%X5 := FALSE;
   "HMI_DB".Drives.Drive_3UZ1.Alarms.AlarmsWord4.%X6 := FALSE;
   "HMI_DB".Drives.Drive_3UZ1.Alarms.AlarmsWord4.%X7 := FALSE;
   "HMI_DB".Drives.Drive_3UZ1.Alarms.AlarmsWord4.%X8 := FALSE;
   "HMI_DB".Drives.Drive_3UZ1.Alarms.AlarmsWord4.%X9 := FALSE;
   "HMI_DB".Drives.Drive_3UZ1.Alarms.AlarmsWord4.%X10 := FALSE;
   "HMI_DB".Drives.Drive_3UZ1.Alarms.AlarmsWord4.%X11 := FALSE;
   "HMI_DB".Drives.Drive_3UZ1.Alarms.AlarmsWord4.%X12 := FALSE;
   "HMI_DB".Drives.Drive_3UZ1.Alarms.AlarmsWord4.%X13 := FALSE;
   "HMI_DB".Drives.Drive_3UZ1.Alarms.AlarmsWord4.%X14 := FALSE;
   "HMI_DB".Drives.Drive_3UZ1.Alarms.AlarmsWord4.%X15 := FALSE;
END_REGION

REGION Network 4 (SCL): Формування слів попереджень для HMI - ПЧ 4UZ1
   // ============================================================
   // 1. AlarmsWord1
   // ============================================================

   "HMI_DB".Drives.Drive_4UZ1.Alarms.AlarmsWord1.%X0 := "DB_Drive_4UZ1".Status.%X5 AND ("DB_Drive_4UZ1".WarningCode = W#16#0636); // A01590
   "HMI_DB".Drives.Drive_4UZ1.Alarms.AlarmsWord1.%X1 := "DB_Drive_4UZ1".Status.%X5 AND ("DB_Drive_4UZ1".WarningCode = W#16#0682); // A01666
   "HMI_DB".Drives.Drive_4UZ1.Alarms.AlarmsWord1.%X2 := "DB_Drive_4UZ1".Status.%X5 AND ("DB_Drive_4UZ1".WarningCode = W#16#06A2); // A01698
   "HMI_DB".Drives.Drive_4UZ1.Alarms.AlarmsWord1.%X3 := "DB_Drive_4UZ1".Status.%X5 AND ("DB_Drive_4UZ1".WarningCode = W#16#06A3); // A01699
   "HMI_DB".Drives.Drive_4UZ1.Alarms.AlarmsWord1.%X4 := "DB_Drive_4UZ1".Status.%X5 AND ("DB_Drive_4UZ1".WarningCode = W#16#076C); // A01900
   "HMI_DB".Drives.Drive_4UZ1.Alarms.AlarmsWord1.%X5 := "DB_Drive_4UZ1".Status.%X5 AND ("DB_Drive_4UZ1".WarningCode = W#16#0780); // A01920
   "HMI_DB".Drives.Drive_4UZ1.Alarms.AlarmsWord1.%X6 := "DB_Drive_4UZ1".Status.%X5 AND ("DB_Drive_4UZ1".WarningCode = W#16#1388); // A05000
   "HMI_DB".Drives.Drive_4UZ1.Alarms.AlarmsWord1.%X7 := "DB_Drive_4UZ1".Status.%X5 AND ("DB_Drive_4UZ1".WarningCode = W#16#1389); // A05001
   "HMI_DB".Drives.Drive_4UZ1.Alarms.AlarmsWord1.%X8 := "DB_Drive_4UZ1".Status.%X5 AND ("DB_Drive_4UZ1".WarningCode = W#16#138A); // A05002
   "HMI_DB".Drives.Drive_4UZ1.Alarms.AlarmsWord1.%X9 := "DB_Drive_4UZ1".Status.%X5 AND ("DB_Drive_4UZ1".WarningCode = W#16#138C); // A05004
   "HMI_DB".Drives.Drive_4UZ1.Alarms.AlarmsWord1.%X10 := "DB_Drive_4UZ1".Status.%X5 AND ("DB_Drive_4UZ1".WarningCode = W#16#138E); // A05006
   "HMI_DB".Drives.Drive_4UZ1.Alarms.AlarmsWord1.%X11 := "DB_Drive_4UZ1".Status.%X5 AND ("DB_Drive_4UZ1".WarningCode = W#16#1B64); // A07012
   "HMI_DB".Drives.Drive_4UZ1.Alarms.AlarmsWord1.%X12 := "DB_Drive_4UZ1".Status.%X5 AND ("DB_Drive_4UZ1".WarningCode = W#16#03F5); // A01013
   "HMI_DB".Drives.Drive_4UZ1.Alarms.AlarmsWord1.%X13 := "DB_Drive_4UZ1".Status.%X5 AND ("DB_Drive_4UZ1".WarningCode = W#16#1C99); // A07321
   "HMI_DB".Drives.Drive_4UZ1.Alarms.AlarmsWord1.%X14 := "DB_Drive_4UZ1".Status.%X5 AND ("DB_Drive_4UZ1".WarningCode = W#16#1CE8); // A07400
   "HMI_DB".Drives.Drive_4UZ1.Alarms.AlarmsWord1.%X15 := "DB_Drive_4UZ1".Status.%X5 AND ("DB_Drive_4UZ1".WarningCode = W#16#1CF1); // A07409

   // ============================================================
   // 2. AlarmsWord2
   // ============================================================

   "HMI_DB".Drives.Drive_4UZ1.Alarms.AlarmsWord2.%X0 := "DB_Drive_4UZ1".Status.%X5 AND ("DB_Drive_4UZ1".WarningCode = W#16#1E7D); // A07805
   "HMI_DB".Drives.Drive_4UZ1.Alarms.AlarmsWord2.%X1 := "DB_Drive_4UZ1".Status.%X5 AND ("DB_Drive_4UZ1".WarningCode = W#16#1EAA); // A07850
   "HMI_DB".Drives.Drive_4UZ1.Alarms.AlarmsWord2.%X2 := "DB_Drive_4UZ1".Status.%X5 AND ("DB_Drive_4UZ1".WarningCode = W#16#1EAB); // A07851
   "HMI_DB".Drives.Drive_4UZ1.Alarms.AlarmsWord2.%X3 := "DB_Drive_4UZ1".Status.%X5 AND ("DB_Drive_4UZ1".WarningCode = W#16#1EAC); // A07852
   "HMI_DB".Drives.Drive_4UZ1.Alarms.AlarmsWord2.%X4 := "DB_Drive_4UZ1".Status.%X5 AND ("DB_Drive_4UZ1".WarningCode = W#16#1EDF); // A07903
   "HMI_DB".Drives.Drive_4UZ1.Alarms.AlarmsWord2.%X5 := "DB_Drive_4UZ1".Status.%X5 AND ("DB_Drive_4UZ1".WarningCode = W#16#1EE6); // A07910
   "HMI_DB".Drives.Drive_4UZ1.Alarms.AlarmsWord2.%X6 := "DB_Drive_4UZ1".Status.%X5 AND ("DB_Drive_4UZ1".WarningCode = W#16#1EF0); // A07920
   "HMI_DB".Drives.Drive_4UZ1.Alarms.AlarmsWord2.%X7 := "DB_Drive_4UZ1".Status.%X5 AND ("DB_Drive_4UZ1".WarningCode = W#16#1EF1); // A07921
   "HMI_DB".Drives.Drive_4UZ1.Alarms.AlarmsWord2.%X8 := "DB_Drive_4UZ1".Status.%X5 AND ("DB_Drive_4UZ1".WarningCode = W#16#1EF2); // A07922
   "HMI_DB".Drives.Drive_4UZ1.Alarms.AlarmsWord2.%X9 := "DB_Drive_4UZ1".Status.%X5 AND ("DB_Drive_4UZ1".WarningCode = W#16#1EF7); // A07927
   "HMI_DB".Drives.Drive_4UZ1.Alarms.AlarmsWord2.%X10 := "DB_Drive_4UZ1".Status.%X5 AND ("DB_Drive_4UZ1".WarningCode = W#16#1F2C); // A07980
   "HMI_DB".Drives.Drive_4UZ1.Alarms.AlarmsWord2.%X11 := "DB_Drive_4UZ1".Status.%X5 AND ("DB_Drive_4UZ1".WarningCode = W#16#1F2D); // A07981
   "HMI_DB".Drives.Drive_4UZ1.Alarms.AlarmsWord2.%X12 := "DB_Drive_4UZ1".Status.%X5 AND ("DB_Drive_4UZ1".WarningCode = W#16#1F37); // A07991
   "HMI_DB".Drives.Drive_4UZ1.Alarms.AlarmsWord2.%X13 := "DB_Drive_4UZ1".Status.%X5 AND ("DB_Drive_4UZ1".WarningCode = W#16#213F); // A08511
   "HMI_DB".Drives.Drive_4UZ1.Alarms.AlarmsWord2.%X14 := "DB_Drive_4UZ1".Status.%X5 AND ("DB_Drive_4UZ1".WarningCode = W#16#214E); // A08526
   "HMI_DB".Drives.Drive_4UZ1.Alarms.AlarmsWord2.%X15 := "DB_Drive_4UZ1".Status.%X5 AND ("DB_Drive_4UZ1".WarningCode = W#16#2175); // A08565


   // ============================================================
   // 3. AlarmsWord3
   // ============================================================

   "HMI_DB".Drives.Drive_4UZ1.Alarms.AlarmsWord3.%X0 := "DB_Drive_4UZ1".Status.%X5 AND ("DB_Drive_4UZ1".WarningCode = W#16#7561); // A30049
   "HMI_DB".Drives.Drive_4UZ1.Alarms.AlarmsWord3.%X1 := "DB_Drive_4UZ1".Status.%X5 AND ("DB_Drive_4UZ1".WarningCode = W#16#7726); // A30502
   "HMI_DB".Drives.Drive_4UZ1.Alarms.AlarmsWord3.%X2 := "DB_Drive_4UZ1".Status.%X5 AND ("DB_Drive_4UZ1".WarningCode = W#16#78C8); // A30920
   "HMI_DB".Drives.Drive_4UZ1.Alarms.AlarmsWord3.%X3 := "DB_Drive_4UZ1".Status.%X5 AND ("DB_Drive_4UZ1".WarningCode = W#16#183D); // A06205
   "HMI_DB".Drives.Drive_4UZ1.Alarms.AlarmsWord3.%X4 := "DB_Drive_4UZ1".Status.%X5 AND ("DB_Drive_4UZ1".WarningCode = W#16#183E); // A06206
   "HMI_DB".Drives.Drive_4UZ1.Alarms.AlarmsWord3.%X5 := "DB_Drive_4UZ1".Status.%X5 AND ("DB_Drive_4UZ1".WarningCode = W#16#1840); // A06208
   "HMI_DB".Drives.Drive_4UZ1.Alarms.AlarmsWord3.%X6 := "DB_Drive_4UZ1".Status.%X5 AND ("DB_Drive_4UZ1".WarningCode = W#16#1847); // A06215
   "HMI_DB".Drives.Drive_4UZ1.Alarms.AlarmsWord3.%X7 := "DB_Drive_4UZ1".Status.%X5 AND ("DB_Drive_4UZ1".WarningCode = W#16#186A); // A06250
   "HMI_DB".Drives.Drive_4UZ1.Alarms.AlarmsWord3.%X8 := "DB_Drive_4UZ1".Status.%X5 AND ("DB_Drive_4UZ1".WarningCode = W#16#1874); // A06260
   "HMI_DB".Drives.Drive_4UZ1.Alarms.AlarmsWord3.%X9 := "DB_Drive_4UZ1".Status.%X5 AND ("DB_Drive_4UZ1".WarningCode = W#16#189D); // A06301
   "HMI_DB".Drives.Drive_4UZ1.Alarms.AlarmsWord3.%X10 := "DB_Drive_4UZ1".Status.%X5 AND ("DB_Drive_4UZ1".WarningCode = W#16#18CE); // A06350
   "HMI_DB".Drives.Drive_4UZ1.Alarms.AlarmsWord3.%X11 := "DB_Drive_4UZ1".Status.%X5 AND ("DB_Drive_4UZ1".WarningCode = W#16#18CF); // A06351
   "HMI_DB".Drives.Drive_4UZ1.Alarms.AlarmsWord3.%X12 := "DB_Drive_4UZ1".Status.%X5 AND ("DB_Drive_4UZ1".WarningCode = W#16#1A90); // A06800
   "HMI_DB".Drives.Drive_4UZ1.Alarms.AlarmsWord3.%X13 := "DB_Drive_4UZ1".Status.%X5 AND ("DB_Drive_4UZ1".WarningCode = W#16#7552); // A30034
   "HMI_DB".Drives.Drive_4UZ1.Alarms.AlarmsWord3.%X14 := "DB_Drive_4UZ1".Status.%X5 AND ("DB_Drive_4UZ1".WarningCode = W#16#7559); // A30041
   "HMI_DB".Drives.Drive_4UZ1.Alarms.AlarmsWord3.%X15 := "DB_Drive_4UZ1".Status.%X5 AND ("DB_Drive_4UZ1".WarningCode = W#16#755A); // A30042


   // ============================================================
   // 4. AlarmsWord4
   // ============================================================

   "HMI_DB".Drives.Drive_4UZ1.Alarms.AlarmsWord4.%X0 := "DB_Drive_4UZ1".Status.%X5 AND ("DB_Drive_4UZ1".WarningCode = W#16#755C); // A30044
   "HMI_DB".Drives.Drive_4UZ1.Alarms.AlarmsWord4.%X1 := "DB_Drive_4UZ1".Status.%X5 AND ("DB_Drive_4UZ1".WarningCode = W#16#755E); // A30046
   "HMI_DB".Drives.Drive_4UZ1.Alarms.AlarmsWord4.%X2 := "DB_Drive_4UZ1".Status.%X5 AND ("DB_Drive_4UZ1".WarningCode = W#16#757D); // A30077
   "HMI_DB".Drives.Drive_4UZ1.Alarms.AlarmsWord4.%X3 := "DB_Drive_4UZ1".Status.%X5 AND ("DB_Drive_4UZ1".WarningCode = W#16#757F); // A30079

   // Невикористані біти
   "HMI_DB".Drives.Drive_4UZ1.Alarms.AlarmsWord4.%X4 := FALSE;
   "HMI_DB".Drives.Drive_4UZ1.Alarms.AlarmsWord4.%X5 := FALSE;
   "HMI_DB".Drives.Drive_4UZ1.Alarms.AlarmsWord4.%X6 := FALSE;
   "HMI_DB".Drives.Drive_4UZ1.Alarms.AlarmsWord4.%X7 := FALSE;
   "HMI_DB".Drives.Drive_4UZ1.Alarms.AlarmsWord4.%X8 := FALSE;
   "HMI_DB".Drives.Drive_4UZ1.Alarms.AlarmsWord4.%X9 := FALSE;
   "HMI_DB".Drives.Drive_4UZ1.Alarms.AlarmsWord4.%X10 := FALSE;
   "HMI_DB".Drives.Drive_4UZ1.Alarms.AlarmsWord4.%X11 := FALSE;
   "HMI_DB".Drives.Drive_4UZ1.Alarms.AlarmsWord4.%X12 := FALSE;
   "HMI_DB".Drives.Drive_4UZ1.Alarms.AlarmsWord4.%X13 := FALSE;
   "HMI_DB".Drives.Drive_4UZ1.Alarms.AlarmsWord4.%X14 := FALSE;
   "HMI_DB".Drives.Drive_4UZ1.Alarms.AlarmsWord4.%X15 := FALSE;
END_REGION

REGION Network 5 (SCL): Формування слів попереджень для HMI - ПЧ 4UZ2
   // ============================================================
   // 1. AlarmsWord1
   // ============================================================

   "HMI_DB".Drives.Drive_4UZ2.Alarms.AlarmsWord1.%X0 := "DB_Drive_4UZ2".Status.%X5 AND ("DB_Drive_4UZ2".WarningCode = W#16#0636); // A01590
   "HMI_DB".Drives.Drive_4UZ2.Alarms.AlarmsWord1.%X1 := "DB_Drive_4UZ2".Status.%X5 AND ("DB_Drive_4UZ2".WarningCode = W#16#0682); // A01666
   "HMI_DB".Drives.Drive_4UZ2.Alarms.AlarmsWord1.%X2 := "DB_Drive_4UZ2".Status.%X5 AND ("DB_Drive_4UZ2".WarningCode = W#16#06A2); // A01698
   "HMI_DB".Drives.Drive_4UZ2.Alarms.AlarmsWord1.%X3 := "DB_Drive_4UZ2".Status.%X5 AND ("DB_Drive_4UZ2".WarningCode = W#16#06A3); // A01699
   "HMI_DB".Drives.Drive_4UZ2.Alarms.AlarmsWord1.%X4 := "DB_Drive_4UZ2".Status.%X5 AND ("DB_Drive_4UZ2".WarningCode = W#16#076C); // A01900
   "HMI_DB".Drives.Drive_4UZ2.Alarms.AlarmsWord1.%X5 := "DB_Drive_4UZ2".Status.%X5 AND ("DB_Drive_4UZ2".WarningCode = W#16#0780); // A01920
   "HMI_DB".Drives.Drive_4UZ2.Alarms.AlarmsWord1.%X6 := "DB_Drive_4UZ2".Status.%X5 AND ("DB_Drive_4UZ2".WarningCode = W#16#1388); // A05000
   "HMI_DB".Drives.Drive_4UZ2.Alarms.AlarmsWord1.%X7 := "DB_Drive_4UZ2".Status.%X5 AND ("DB_Drive_4UZ2".WarningCode = W#16#1389); // A05001
   "HMI_DB".Drives.Drive_4UZ2.Alarms.AlarmsWord1.%X8 := "DB_Drive_4UZ2".Status.%X5 AND ("DB_Drive_4UZ2".WarningCode = W#16#138A); // A05002
   "HMI_DB".Drives.Drive_4UZ2.Alarms.AlarmsWord1.%X9 := "DB_Drive_4UZ2".Status.%X5 AND ("DB_Drive_4UZ2".WarningCode = W#16#138C); // A05004
   "HMI_DB".Drives.Drive_4UZ2.Alarms.AlarmsWord1.%X10 := "DB_Drive_4UZ2".Status.%X5 AND ("DB_Drive_4UZ2".WarningCode = W#16#138E); // A05006
   "HMI_DB".Drives.Drive_4UZ2.Alarms.AlarmsWord1.%X11 := "DB_Drive_4UZ2".Status.%X5 AND ("DB_Drive_4UZ2".WarningCode = W#16#1B64); // A07012
   "HMI_DB".Drives.Drive_4UZ2.Alarms.AlarmsWord1.%X12 := "DB_Drive_4UZ2".Status.%X5 AND ("DB_Drive_4UZ2".WarningCode = W#16#03F5); // A01013
   "HMI_DB".Drives.Drive_4UZ2.Alarms.AlarmsWord1.%X13 := "DB_Drive_4UZ2".Status.%X5 AND ("DB_Drive_4UZ2".WarningCode = W#16#1C99); // A07321
   "HMI_DB".Drives.Drive_4UZ2.Alarms.AlarmsWord1.%X14 := "DB_Drive_4UZ2".Status.%X5 AND ("DB_Drive_4UZ2".WarningCode = W#16#1CE8); // A07400
   "HMI_DB".Drives.Drive_4UZ2.Alarms.AlarmsWord1.%X15 := "DB_Drive_4UZ2".Status.%X5 AND ("DB_Drive_4UZ2".WarningCode = W#16#1CF1); // A07409

   // ============================================================
   // 2. AlarmsWord2
   // ============================================================

   "HMI_DB".Drives.Drive_4UZ2.Alarms.AlarmsWord2.%X0 := "DB_Drive_4UZ2".Status.%X5 AND ("DB_Drive_4UZ2".WarningCode = W#16#1E7D); // A07805
   "HMI_DB".Drives.Drive_4UZ2.Alarms.AlarmsWord2.%X1 := "DB_Drive_4UZ2".Status.%X5 AND ("DB_Drive_4UZ2".WarningCode = W#16#1EAA); // A07850
   "HMI_DB".Drives.Drive_4UZ2.Alarms.AlarmsWord2.%X2 := "DB_Drive_4UZ2".Status.%X5 AND ("DB_Drive_4UZ2".WarningCode = W#16#1EAB); // A07851
   "HMI_DB".Drives.Drive_4UZ2.Alarms.AlarmsWord2.%X3 := "DB_Drive_4UZ2".Status.%X5 AND ("DB_Drive_4UZ2".WarningCode = W#16#1EAC); // A07852
   "HMI_DB".Drives.Drive_4UZ2.Alarms.AlarmsWord2.%X4 := "DB_Drive_4UZ2".Status.%X5 AND ("DB_Drive_4UZ2".WarningCode = W#16#1EDF); // A07903
   "HMI_DB".Drives.Drive_4UZ2.Alarms.AlarmsWord2.%X5 := "DB_Drive_4UZ2".Status.%X5 AND ("DB_Drive_4UZ2".WarningCode = W#16#1EE6); // A07910
   "HMI_DB".Drives.Drive_4UZ2.Alarms.AlarmsWord2.%X6 := "DB_Drive_4UZ2".Status.%X5 AND ("DB_Drive_4UZ2".WarningCode = W#16#1EF0); // A07920
   "HMI_DB".Drives.Drive_4UZ2.Alarms.AlarmsWord2.%X7 := "DB_Drive_4UZ2".Status.%X5 AND ("DB_Drive_4UZ2".WarningCode = W#16#1EF1); // A07921
   "HMI_DB".Drives.Drive_4UZ2.Alarms.AlarmsWord2.%X8 := "DB_Drive_4UZ2".Status.%X5 AND ("DB_Drive_4UZ2".WarningCode = W#16#1EF2); // A07922
   "HMI_DB".Drives.Drive_4UZ2.Alarms.AlarmsWord2.%X9 := "DB_Drive_4UZ2".Status.%X5 AND ("DB_Drive_4UZ2".WarningCode = W#16#1EF7); // A07927
   "HMI_DB".Drives.Drive_4UZ2.Alarms.AlarmsWord2.%X10 := "DB_Drive_4UZ2".Status.%X5 AND ("DB_Drive_4UZ2".WarningCode = W#16#1F2C); // A07980
   "HMI_DB".Drives.Drive_4UZ2.Alarms.AlarmsWord2.%X11 := "DB_Drive_4UZ2".Status.%X5 AND ("DB_Drive_4UZ2".WarningCode = W#16#1F2D); // A07981
   "HMI_DB".Drives.Drive_4UZ2.Alarms.AlarmsWord2.%X12 := "DB_Drive_4UZ2".Status.%X5 AND ("DB_Drive_4UZ2".WarningCode = W#16#1F37); // A07991
   "HMI_DB".Drives.Drive_4UZ2.Alarms.AlarmsWord2.%X13 := "DB_Drive_4UZ2".Status.%X5 AND ("DB_Drive_4UZ2".WarningCode = W#16#213F); // A08511
   "HMI_DB".Drives.Drive_4UZ2.Alarms.AlarmsWord2.%X14 := "DB_Drive_4UZ2".Status.%X5 AND ("DB_Drive_4UZ2".WarningCode = W#16#214E); // A08526
   "HMI_DB".Drives.Drive_4UZ2.Alarms.AlarmsWord2.%X15 := "DB_Drive_4UZ2".Status.%X5 AND ("DB_Drive_4UZ2".WarningCode = W#16#2175); // A08565


   // ============================================================
   // 3. AlarmsWord3
   // ============================================================

   "HMI_DB".Drives.Drive_4UZ2.Alarms.AlarmsWord3.%X0 := "DB_Drive_4UZ2".Status.%X5 AND ("DB_Drive_4UZ2".WarningCode = W#16#7561); // A30049
   "HMI_DB".Drives.Drive_4UZ2.Alarms.AlarmsWord3.%X1 := "DB_Drive_4UZ2".Status.%X5 AND ("DB_Drive_4UZ2".WarningCode = W#16#7726); // A30502
   "HMI_DB".Drives.Drive_4UZ2.Alarms.AlarmsWord3.%X2 := "DB_Drive_4UZ2".Status.%X5 AND ("DB_Drive_4UZ2".WarningCode = W#16#78C8); // A30920
   "HMI_DB".Drives.Drive_4UZ2.Alarms.AlarmsWord3.%X3 := "DB_Drive_4UZ2".Status.%X5 AND ("DB_Drive_4UZ2".WarningCode = W#16#183D); // A06205
   "HMI_DB".Drives.Drive_4UZ2.Alarms.AlarmsWord3.%X4 := "DB_Drive_4UZ2".Status.%X5 AND ("DB_Drive_4UZ2".WarningCode = W#16#183E); // A06206
   "HMI_DB".Drives.Drive_4UZ2.Alarms.AlarmsWord3.%X5 := "DB_Drive_4UZ2".Status.%X5 AND ("DB_Drive_4UZ2".WarningCode = W#16#1840); // A06208
   "HMI_DB".Drives.Drive_4UZ2.Alarms.AlarmsWord3.%X6 := "DB_Drive_4UZ2".Status.%X5 AND ("DB_Drive_4UZ2".WarningCode = W#16#1847); // A06215
   "HMI_DB".Drives.Drive_4UZ2.Alarms.AlarmsWord3.%X7 := "DB_Drive_4UZ2".Status.%X5 AND ("DB_Drive_4UZ2".WarningCode = W#16#186A); // A06250
   "HMI_DB".Drives.Drive_4UZ2.Alarms.AlarmsWord3.%X8 := "DB_Drive_4UZ2".Status.%X5 AND ("DB_Drive_4UZ2".WarningCode = W#16#1874); // A06260
   "HMI_DB".Drives.Drive_4UZ2.Alarms.AlarmsWord3.%X9 := "DB_Drive_4UZ2".Status.%X5 AND ("DB_Drive_4UZ2".WarningCode = W#16#189D); // A06301
   "HMI_DB".Drives.Drive_4UZ2.Alarms.AlarmsWord3.%X10 := "DB_Drive_4UZ2".Status.%X5 AND ("DB_Drive_4UZ2".WarningCode = W#16#18CE); // A06350
   "HMI_DB".Drives.Drive_4UZ2.Alarms.AlarmsWord3.%X11 := "DB_Drive_4UZ2".Status.%X5 AND ("DB_Drive_4UZ2".WarningCode = W#16#18CF); // A06351
   "HMI_DB".Drives.Drive_4UZ2.Alarms.AlarmsWord3.%X12 := "DB_Drive_4UZ2".Status.%X5 AND ("DB_Drive_4UZ2".WarningCode = W#16#1A90); // A06800
   "HMI_DB".Drives.Drive_4UZ2.Alarms.AlarmsWord3.%X13 := "DB_Drive_4UZ2".Status.%X5 AND ("DB_Drive_4UZ2".WarningCode = W#16#7552); // A30034
   "HMI_DB".Drives.Drive_4UZ2.Alarms.AlarmsWord3.%X14 := "DB_Drive_4UZ2".Status.%X5 AND ("DB_Drive_4UZ2".WarningCode = W#16#7559); // A30041
   "HMI_DB".Drives.Drive_4UZ2.Alarms.AlarmsWord3.%X15 := "DB_Drive_4UZ2".Status.%X5 AND ("DB_Drive_4UZ2".WarningCode = W#16#755A); // A30042


   // ============================================================
   // 4. AlarmsWord4
   // ============================================================

   "HMI_DB".Drives.Drive_4UZ2.Alarms.AlarmsWord4.%X0 := "DB_Drive_4UZ2".Status.%X5 AND ("DB_Drive_4UZ2".WarningCode = W#16#755C); // A30044
   "HMI_DB".Drives.Drive_4UZ2.Alarms.AlarmsWord4.%X1 := "DB_Drive_4UZ2".Status.%X5 AND ("DB_Drive_4UZ2".WarningCode = W#16#755E); // A30046
   "HMI_DB".Drives.Drive_4UZ2.Alarms.AlarmsWord4.%X2 := "DB_Drive_4UZ2".Status.%X5 AND ("DB_Drive_4UZ2".WarningCode = W#16#757D); // A30077
   "HMI_DB".Drives.Drive_4UZ2.Alarms.AlarmsWord4.%X3 := "DB_Drive_4UZ2".Status.%X5 AND ("DB_Drive_4UZ2".WarningCode = W#16#757F); // A30079

   // Невикористані біти
   "HMI_DB".Drives.Drive_4UZ2.Alarms.AlarmsWord4.%X4 := FALSE;
   "HMI_DB".Drives.Drive_4UZ2.Alarms.AlarmsWord4.%X5 := FALSE;
   "HMI_DB".Drives.Drive_4UZ2.Alarms.AlarmsWord4.%X6 := FALSE;
   "HMI_DB".Drives.Drive_4UZ2.Alarms.AlarmsWord4.%X7 := FALSE;
   "HMI_DB".Drives.Drive_4UZ2.Alarms.AlarmsWord4.%X8 := FALSE;
   "HMI_DB".Drives.Drive_4UZ2.Alarms.AlarmsWord4.%X9 := FALSE;
   "HMI_DB".Drives.Drive_4UZ2.Alarms.AlarmsWord4.%X10 := FALSE;
   "HMI_DB".Drives.Drive_4UZ2.Alarms.AlarmsWord4.%X11 := FALSE;
   "HMI_DB".Drives.Drive_4UZ2.Alarms.AlarmsWord4.%X12 := FALSE;
   "HMI_DB".Drives.Drive_4UZ2.Alarms.AlarmsWord4.%X13 := FALSE;
   "HMI_DB".Drives.Drive_4UZ2.Alarms.AlarmsWord4.%X14 := FALSE;
   "HMI_DB".Drives.Drive_4UZ2.Alarms.AlarmsWord4.%X15 := FALSE;
END_REGION
END_FUNCTION

// folder: 600_Diagnostic

FUNCTION_BLOCK "FB_Diag_MRP"   // FB601, SCL
{ S7_Optimized_Access := 'TRUE' }
VERSION : 1.0
// FB601. Комплексна діагностика PROFINET та кільця MRP. Окремо визначає наявність IO-пристроїв, достовірність діагностики, стан кільця за даними менеджера та стан чотирьох фізичних ділянок. Викликається через FC614; дані й мультиекземпляри зберігаються у DB630.
   VAR_INPUT
      IO_System : Hw_IoSystem;   // Апаратний ідентифікатор системи PROFINET IO; не ідентифікатор окремого порту або привода.
   END_VAR
   VAR_OUTPUT
      Alarm_Ring_Broken_Scalance : Bool;   // Сумісна ознака: підтверджений обрив принаймні однієї з двох ділянок біля SCALANCE.
      Alarm_Ring_Broken_Drive : Bool;   // Сумісна ознака: підтверджений обрив принаймні однієї з двох ділянок біля CU привода.
      Alarm_Ring_Broken_HMI : Bool;   // Сумісна ознака: підтверджений обрив принаймні однієї з двох ділянок біля HMI.
      Alarm_Station_Drive_Offline : Bool;   // Привод №1 відсутній за достовірними даними після пускової витримки 10 с.
      Alarm_Station_HMI_Offline : Bool;   // HMI №7 відсутня як IO-пристрій за достовірними даними після пускової витримки 10 с.
      Ring_Ok : Bool;   // Менеджер достовірно повідомляє про замкнене кільце; це не ознака справності всіх модулів.
      Ring_StateValid : Bool;   // Отримано придатний і достатньо свіжий запис стану кільця від менеджера.
      Ring_Open : Bool;   // Менеджер достовірно повідомляє про розімкнене кільце.
      Diagnostics_Valid : Bool;   // Достовірні дані системи IO, вузлів, менеджера та всіх чотирьох фізичних ділянок.
      Diagnostics_Unknown : Bool;   // Недостовірність триває 5 с і минула пускова витримка 10 с. Це окремий сервісний прапорець.
      Ring_Open_Unlocalized : Bool;   // Кільце достовірно розімкнене, але жодна ділянка не має підтвердженої відфільтрованої ознаки обриву.
      DeviceStates_Valid : Bool;   // Обидва виклики DeviceStates завершилися з кодом 0.
      HMI_StatusValid : Bool;   // Достовірність перевірки наявності HMI як IO-пристрою.
      HMI_IO_Online : Bool;   // IO-пристрій HMI №7 присутній; не замінює перевірку сигналу життя.
      HMI_CommunicationFault : Bool;   // Після 10 с пуску немає HMI як IO-пристрою або відсутній її сигнал життя.
      Nodes_Valid : Bool;   // Достовірність діагностики ПЛК, SCALANCE, привода та чотирьох енкодерів.
      DisplayUnknown : Bool;   // Негайна жовта індикація HMI: принаймні одне необхідне джерело даних недостовірне.
      DisplayOpen : Bool;   // Індикація HMI про підтверджене розімкнене кільце.
      DisplayClosed : Bool;   // Індикація HMI про підтверджене замкнене кільце.
      DisplayHmiNoFault : Bool;   // Повідомлення про звʼязок HMI, якщо інші діагностичні дані достовірні; інакше показується невідомий стан.
      Scalance_Online : Bool;   // Достовірна наявність SCALANCE №2; дозволяє опитування його портів.
      Drive_Online : Bool;   // Достовірна наявність привода №1; дозволяє опитування його портів.
      Alarm_Station_Scalance_Offline : Bool;   // SCALANCE №2 відсутній за достовірними даними після пускової витримки 10 с.
      Segment_PLC_HMI_Valid : Bool;   // Для ділянки PLC_HMI доступний принаймні один достовірний стан фізичного порту.
      Segment_PLC_SCALANCE_Valid : Bool;   // Для ділянки PLC_SCALANCE доступний принаймні один достовірний стан фізичного порту.
      Segment_SCALANCE_CU_Valid : Bool;   // Для ділянки SCALANCE_CU доступний принаймні один достовірний стан фізичного порту.
      Segment_HMI_CU_Valid : Bool;   // Для ділянки HMI_CU доступний принаймні один достовірний стан фізичного порту.
      Segment_PLC_HMI_Down : Bool;   // Підтверджений фізичний Link Down ділянки PLC_HMI після фільтра 1 с; джерело відповідного хрестика HMI.
      Segment_PLC_SCALANCE_Down : Bool;   // Підтверджений фізичний Link Down ділянки PLC_SCALANCE після фільтра 1 с; джерело відповідного хрестика HMI.
      Segment_SCALANCE_CU_Down : Bool;   // Підтверджений фізичний Link Down ділянки SCALANCE_CU після фільтра 1 с; джерело відповідного хрестика HMI.
      Segment_HMI_CU_Down : Bool;   // Підтверджений фізичний Link Down ділянки HMI_CU після фільтра 1 с; джерело відповідного хрестика HMI.
   END_VAR
   VAR
      DeviceProblems : Array[0..1023] of Bool;   // Повний буфер 1024 біт для DeviceStates MODE 5; не є маскою обривів портів.
      DevicePresence : Array[0..1023] of Bool;   // Повний буфер 1024 біт для DeviceStates MODE 4. Біт n відповідає номеру IO-пристрою n.
      Manager : "FB_MRP_RecordReader";   // Мультиекземпляр FB615 для читання запису менеджера MRP з інтерфейсу ПЛК.
      PlcP1 : "FB_MRP_RecordReader";   // Мультиекземпляр FB615 для фізичного порту PLC X1 P1, ділянка PLC—HMI.
      PlcP2 : "FB_MRP_RecordReader";   // Мультиекземпляр FB615 для фізичного порту PLC X1 P2, ділянка PLC—SCALANCE.
      SwitchP5 : "FB_MRP_RecordReader";   // Мультиекземпляр FB615 для порту SCALANCE P5, ділянка PLC—SCALANCE.
      SwitchP7 : "FB_MRP_RecordReader";   // Мультиекземпляр FB615 для порту SCALANCE P7, ділянка SCALANCE—CU.
      DriveP1 : "FB_MRP_RecordReader";   // Мультиекземпляр FB615 для порту CU P1, ділянка SCALANCE—CU.
      DriveP2 : "FB_MRP_RecordReader";   // Мультиекземпляр FB615 для порту CU P2, ділянка HMI—CU.
      Startup : TON_TIME;   // Пускова витримка 10 с для сигналів відсутності станцій та звʼязку HMI.
      BadDiagnostics : TON_TIME;   // Витримка 5 с перед установленням сервісної ознаки недостовірної діагностики.
      LinkAlarm1 : TON_TIME;   // Фільтр 1 с для підтвердженого Link Down ділянки PLC—HMI.
      LinkAlarm2 : TON_TIME;   // Фільтр 1 с для підтвердженого Link Down ділянки PLC—SCALANCE.
      LinkAlarm3 : TON_TIME;   // Фільтр 1 с для підтвердженого Link Down ділянки SCALANCE—CU.
      LinkAlarm4 : TON_TIME;   // Фільтр 1 с для підтвердженого Link Down ділянки HMI—CU.
   END_VAR
   VAR_TEMP
      anyDown : Bool;   // Принаймні одна ділянка має відфільтровану ознаку фізичного обриву.
      deviceIndex : Int;   // Індекс копіювання перших 128 біт у наявні масиви Data_base без зміни їхнього розміру.
   END_VAR
BEGIN
   // FB601. Комплексна діагностика PROFINET та кільця MRP. Окремо визначає наявність IO-пристроїв, достовірність діагностики, стан кільця за даними менеджера та стан чотирьох фізичних ділянок. Викликається через FC614; дані й мультиекземпляри зберігаються у DB630.
   // Викликати циклічно після оновлення діагностики вузлів і сигналу життя HMI у FC600.
   // Наявність пристроїв не доводить замкненість кільця; загальна несправність пристрою не визначає обрив кабелю.
   // Червоні хрестики формуються лише за достовірним Link Down. Неотримані або непідтримувані записи означають невідомий стан.

       // 1. Пускова витримка 10 с для повідомлень про відсутність станцій і сигналу життя HMI.
   #Startup(IN := TRUE, PT := T#10s);
       "Data_base".Devices_val_1 := // 2. MODE 5 читає загальні проблеми, MODE 4 — наявність пристроїв. Буфери мають 1024 біти; коди повернення перевіряються.
   DeviceStates(LADDR := #IO_System, MODE := 5,
                                                STATE := #DeviceProblems);
       "Data_base".Devices_val_2 := DeviceStates(LADDR := #IO_System, MODE := 4,
                                                STATE := #DevicePresence);
       // Дані системи IO вважаються достовірними лише після успішного виконання обох запитів.
   #DeviceStates_Valid := ("Data_base".Devices_val_1 = 0) AND ("Data_base".Devices_val_2 = 0);


       FOR #deviceIndex := 0 TO 127 DO
           "Data_base".Devices_With_Errors[#deviceIndex] := ("Data_base".Devices_val_1 = 0) AND #DeviceProblems[#deviceIndex];
           "Data_base".Devices_Online[#deviceIndex] := ("Data_base".Devices_val_2 = 0) AND #DevicePresence[#deviceIndex];
       END_FOR;
       // 3. Номери IO-пристроїв цієї конфігурації: привод — 1, SCALANCE — 2, HMI — 7. У публічні масиви копіюється перевірений префікс без зміни структури Data_base.
   #Drive_Online := #DeviceStates_Valid AND "Data_base".Devices_Online[1];
       #Scalance_Online := #DeviceStates_Valid AND "Data_base".Devices_Online[2];
       "Data_base".Drive_Online := #Drive_Online;

       // Наявність HMI як IO-пристрою та його сигнал життя перевіряються окремо. HMI_Online оновлює мережа 23 FC600.
   #HMI_StatusValid := #DeviceStates_Valid;
       #HMI_IO_Online := #DeviceStates_Valid AND "Data_base".Devices_Online[7];
       #Alarm_Station_HMI_Offline := #Startup.Q AND #HMI_StatusValid AND NOT #HMI_IO_Online;
       #HMI_CommunicationFault := #Startup.Q AND (#Alarm_Station_HMI_Offline OR NOT "Data_base".HMI_Online);
       #Alarm_Station_Drive_Offline := #Startup.Q AND #DeviceStates_Valid AND NOT #Drive_Online;
       #Alarm_Station_Scalance_Offline := #Startup.Q AND #DeviceStates_Valid AND NOT #Scalance_Online;

       // 4. Менеджер: запис 16#8050 з інтерфейсу ПЛК. Порти: запис 16#802A; штатне блокування передавання MRP не є фізичним обривом.
   #Manager(Enable := TRUE, HardwareId := "Local~PROFINET_interface_1", IsRing := TRUE, ExpectedSubslot := 0);
       #PlcP1(Enable := TRUE, HardwareId := "Local~PROFINET_interface_1~Port_1", IsRing := FALSE, ExpectedSubslot := UINT#16#8001);
       #PlcP2(Enable := TRUE, HardwareId := "Local~PROFINET_interface_1~Port_2", IsRing := FALSE, ExpectedSubslot := UINT#16#8002);
       #SwitchP5(Enable := #Scalance_Online, HardwareId := "A1_6~SCALANCE_interface_1~Port_5", IsRing := FALSE, ExpectedSubslot := UINT#16#8005);
       #SwitchP7(Enable := #Scalance_Online, HardwareId := "A1_6~SCALANCE_interface_1~Port_7", IsRing := FALSE, ExpectedSubslot := UINT#16#8007);
       #DriveP1(Enable := #Drive_Online, HardwareId := "Drive_unit_1~PROFINET_interface~Port_1", IsRing := FALSE, ExpectedSubslot := UINT#16#8001);
       #DriveP2(Enable := #Drive_Online, HardwareId := "Drive_unit_1~PROFINET_interface~Port_2", IsRing := FALSE, ExpectedSubslot := UINT#16#8002);

       // 5. Стан кільця береться лише з достовірного запису менеджера. Ring_Status: 1 — замкнене, 0 — розімкнене, -1 — невідомо.
   #Ring_StateValid := #Manager.Valid;
       #Ring_Ok := #Ring_StateValid AND #Manager.UpOrClosed;
       #Ring_Open := #Ring_StateValid AND #Manager.DownOrOpen;
       "Data_base".Ring_Ok := #Ring_Ok;
       IF #Ring_StateValid THEN
           IF #Ring_Ok THEN "Data_base".Ring_Status := 1; ELSE "Data_base".Ring_Status := 0; END_IF;
       ELSE
           "Data_base".Ring_Status := -1;
       END_IF;



       // 6. Ділянки: PLC P1—HMI P1; PLC P2—SC P5; SC P7—CU P1; CU P2—HMI P2. Для двобічної перевірки достатньо одного достовірного кінця.
   #Segment_PLC_HMI_Valid := #PlcP1.Valid;
       #Segment_PLC_SCALANCE_Valid := #PlcP2.Valid OR #SwitchP5.Valid;
       #Segment_SCALANCE_CU_Valid := #SwitchP7.Valid OR #DriveP1.Valid;
       #Segment_HMI_CU_Valid := #DriveP2.Valid;
       // 7. Link Down від доступного кінця має тривати 1 с. Недостовірні дані не запускають таймер; відключення станції саме по собі не визначає ділянку.
   #LinkAlarm1(IN := #PlcP1.Valid AND #PlcP1.DownOrOpen, PT := T#1s);
       #LinkAlarm2(IN := (#PlcP2.Valid AND #PlcP2.DownOrOpen) OR (#SwitchP5.Valid AND #SwitchP5.DownOrOpen), PT := T#1s);
       #LinkAlarm3(IN := (#SwitchP7.Valid AND #SwitchP7.DownOrOpen) OR (#DriveP1.Valid AND #DriveP1.DownOrOpen), PT := T#1s);
       #LinkAlarm4(IN := #DriveP2.Valid AND #DriveP2.DownOrOpen, PT := T#1s);
       #Segment_PLC_HMI_Down := #LinkAlarm1.Q;
       #Segment_PLC_SCALANCE_Down := #LinkAlarm2.Q;
       #Segment_SCALANCE_CU_Down := #LinkAlarm3.Q;
       #Segment_HMI_CU_Down := #LinkAlarm4.Q;
       // Кільце може бути підтверджено розімкненим, хоча конкретну ділянку визначити неможливо. Для цього є Ring_Open_Unlocalized.
   #anyDown := #Segment_PLC_HMI_Down OR #Segment_PLC_SCALANCE_Down OR #Segment_SCALANCE_CU_Down OR #Segment_HMI_CU_Down;
       #Ring_Open_Unlocalized := #Ring_Open AND NOT #anyDown;
       // 8. Перевірити достовірність даних усіх контрольованих вузлів. Достовірність означає наявність придатних даних, а не відсутність несправностей.
   #Nodes_Valid := "DB_DIAG_NODE".DiagnosticsValid AND "FB_DIAG_SCALANCE_NODE_DB".DiagnosticsValid AND
           "DB_DIAG_CU320_NODE".DiagnosticsValid AND "DB_DIAG_ENC_1BR_NODE".DiagnosticsValid AND
           "DB_DIAG_ENC_3BR_NODE".DiagnosticsValid AND "DB_DIAG_ENC_4BR1_NODE".DiagnosticsValid AND
           "DB_DIAG_ENC_4BR2_NODE".DiagnosticsValid;
       #Diagnostics_Valid := #Ring_StateValid AND #DeviceStates_Valid AND #Nodes_Valid AND
                             #Segment_PLC_HMI_Valid AND #Segment_PLC_SCALANCE_Valid AND
                             #Segment_SCALANCE_CU_Valid AND #Segment_HMI_CU_Valid;
       // Сервісний прапорець Diagnostics_Unknown має витримку 5 с та пусковий дозвіл 10 с. Індикація DisplayUnknown зʼявляється одразу за недостовірних даних.
   #BadDiagnostics(IN := NOT #Diagnostics_Valid, PT := T#5s);
       #Diagnostics_Unknown := #Startup.Q AND #BadDiagnostics.Q;
       // 9. Відомий стан кільця може відображатися разом із повідомленням про недоступні інші дані. Невідомий стан має пріоритет над повідомленням HMI на спільному рядку.
   #DisplayUnknown := NOT #Diagnostics_Valid;
       #DisplayOpen := #Ring_Open;
       #DisplayClosed := #Ring_Ok;
       #DisplayHmiNoFault := NOT(#HMI_CommunicationFault);
       // 10. Зберегти сумісні ознаки несправностей біля вузлів. FC614 передає на HMI безпосередньо Segment_*_Down, без старого визначення ділянок за масками пристроїв.
   #Alarm_Ring_Broken_Scalance := #Segment_PLC_SCALANCE_Down OR #Segment_SCALANCE_CU_Down;
       #Alarm_Ring_Broken_Drive := #Segment_SCALANCE_CU_Down OR #Segment_HMI_CU_Down;
       #Alarm_Ring_Broken_HMI := #Segment_PLC_HMI_Down OR #Segment_HMI_CU_Down;
       "Data_base".Alarm_Ring_Broken_Scalance := #Alarm_Ring_Broken_Scalance;
       "Data_base".Alarm_Ring_Broken_Drive := #Alarm_Ring_Broken_Drive;
       "Data_base".Alarm_Ring_Broken_HMI := #Alarm_Ring_Broken_HMI;
       "Data_base".Alarm_Station_Drive_Offline := #Alarm_Station_Drive_Offline;
       "Data_base".Alarm_Station_HMI_Offline := #Alarm_Station_HMI_Offline;
END_FUNCTION_BLOCK

FUNCTION_BLOCK "FB_MRP_RecordReader"   // FB615, SCL
{ S7_Optimized_Access := 'TRUE' }
VERSION : 1.0
// FB615. Асинхронне читання діагностичного запису через RDREC. Кожен екземпляр має власний буфер і таймери. IsRing обирає запис MRP 16#8050 або запис порту 16#802A. Обробляє завершення, помилки, тайм-аут і застарівання даних. Використовується як сім мультиекземплярів у FB601 / DB630.
   VAR_INPUT
      Enable : Bool;   // Дозвіл опитування. FALSE скидає достовірність; активний RDREC продовжує обслуговуватися.
      HardwareId : Hw_Io;   // Апаратний ідентифікатор інтерфейсу менеджера MRP або конкретного фізичного порту.
      IsRing : Bool;   // TRUE: запис MRP 16#8050 і FC613. FALSE: запис порту 16#802A і FC612.
      ExpectedSubslot : UInt;   // Очікуваний підслот фізичного порту, наприклад 16#8001 для порту 1.
   END_VAR
   VAR_OUTPUT
      Valid : Bool;   // Є достовірний, достатньо свіжий результат. Перевіряти разом зі станами й кодом Status.
      UpOrClosed : Bool;   // За Valid=TRUE: фізичний звʼязок встановлено або кільце замкнене, залежно від IsRing.
      DownOrOpen : Bool;   // За Valid=TRUE: фізичний звʼязок відсутній або кільце розімкнене, залежно від IsRing.
      Busy : Bool;   // RDREC виконує асинхронний запит. Це стан виконання, а не ознака несправності.
      Status : DWord;   // Код RDREC або власний код E0010001/2/3. Нуль не замінює перевірку Valid.
      RecordLength : UInt;   // Фактична довжина запису, отримана з виходу LEN інструкції RDREC.
      PortState : Byte;   // Стан передавання/блокування порту з отриманого запису; окремий від фізичного LinkState.
      LinkState : Byte;   // Стан фізичного зʼєднання з отриманого запису. Значення з невизначеним станом не приймаються.
      MrpRole : UInt;   // Роль MRP останнього розібраного запису; оцінювати лише за Valid=TRUE.
   END_VAR
   VAR
      ReadRecord : RDREC;   // Окремий екземпляр RDREC для цього читача.
      Poll : TON_TIME;   // Таймер інтервалу між запитами: 1 секунда.
      Stale : TON_TIME;   // Таймер відсутності нового достовірного результату: 5 секунд.
      Watchdog : TON_TIME;   // Контроль максимальної тривалості очікування активного запиту: 5 секунд.
      Buffer : Array[0..1023] of Byte;   // Власний буфер запису на 1024 байти. Не очищувати й не змінювати під час RDREC.
      Request : Bool;   // Сигнал запуску нового запиту. Повторний запуск заборонено, поки попередній очікується.
      Done : Bool;   // Вихід VALID інструкції RDREC: запис успішно прочитано, але ще потребує перевірки формату.
      Error : Bool;   // Вихід ERROR інструкції RDREC.
      RawStatus : DWord;   // Необроблений код STATUS інструкції RDREC.
      HaveSample : Bool;   // Збережений результат пройшов перевірку і ще може використовуватися.
      Awaiting : Bool;   // Є запит, для якого очікується завершення або помилка.
      readBusy : Bool := FALSE;   // Внутрішнє збереження стану BUSY для керування наступним запитом.
      lastStatus : DWord := DWORD#16#0000_0000;   // Останній діагностичний код, який передається на вихід Status.
   END_VAR
   VAR_TEMP
      Index : DInt;   // Номер запису RDREC, обраний за IsRing.
      NewSample : Bool;   // Ознака нового достовірного результату в поточному циклі; скидає таймер застарівання.
      Parsed : Bool;   // Результат перевірки формату та змісту запису відповідним декодером.
   END_VAR
BEGIN
   // FB615. Асинхронне читання діагностичного запису через RDREC. Кожен екземпляр має власний буфер і таймери. IsRing обирає запис MRP 16#8050 або запис порту 16#802A. Обробляє завершення, помилки, тайм-аут і застарівання даних. Використовується як сім мультиекземплярів у FB601 / DB630.
   // Викликати кожного циклу ПЛК, зокрема поки RDREC зайнятий. HardwareId не змінювати під час запиту.
   // Опитування приблизно раз на секунду; тайм-аут запиту та межа застарівання — 5 секунд.
   // Valid є обовʼязковою умовою використання UpOrClosed / DownOrOpen. Busy не означає несправність.
   // Фільтрація обриву протягом 1 секунди виконується окремо у FB601, а не в цьому читачі.

       #NewSample := FALSE;
       // Запланувати наступне опитування лише за дозволу та вільного RDREC.
   #Poll(IN := #Enable AND NOT #readBusy AND NOT #Request, PT := T#1s);
       #Request := #Poll.Q AND NOT #Awaiting;
       IF #Request THEN #Awaiting := TRUE; END_IF;
       IF #IsRing THEN #Index := DINT#16#8050; ELSE #Index := DINT#16#802A; END_IF;
       // Продовжувати виклик RDREC під час BUSY. Не змінювати й не очищувати його буфер запису.
       #ReadRecord(REQ := #Request, ID := #HardwareId, INDEX := #Index, MLEN := UINT#1024,
                   VALID => #Done, BUSY => #readBusy, ERROR => #Error,
                   STATUS => #RawStatus, LEN => #RecordLength, RECORD := #Buffer);
       // Контролювати час очікування завершення поточного запиту.
   #Watchdog(IN := #Awaiting, PT := T#5s);
       IF #Awaiting AND (#Done OR #Error) THEN
           #Awaiting := FALSE;
           #HaveSample := FALSE;
           IF #Error THEN
               #lastStatus := #RawStatus;
           ELSE
               IF #IsRing THEN
                   #Parsed := "FC_MRP_DecodeRing"(Length := #RecordLength, Data := #Buffer,
                                                  Closed => #UpOrClosed, Role => #MrpRole);
                   #DownOrOpen := #Parsed AND NOT #UpOrClosed;
               ELSE
                   #Parsed := "FC_MRP_DecodePort"(Length := #RecordLength, ExpectedSubslot := #ExpectedSubslot,
                                                  Data := #Buffer, LinkUp => #UpOrClosed, LinkDown => #DownOrOpen,
                                                  PortState => #PortState, LinkState => #LinkState);
               END_IF;
               #HaveSample := #Parsed AND #Enable;
               #NewSample := #HaveSample;
               IF #Parsed THEN #lastStatus := 0; ELSE #lastStatus := DW#16#E0010001; END_IF;
           END_IF;
       END_IF;
       IF #Watchdog.Q THEN
           #HaveSample := FALSE;
           #lastStatus := DW#16#E0010002;
           // Не запускати новий асинхронний запит, доки попередній RDREC не завершився.
           IF NOT #readBusy THEN #Awaiting := FALSE; END_IF;
       END_IF;
       // Новий достовірний результат скидає таймер застарівання.
   #Stale(IN := NOT #NewSample, PT := T#5s);
       IF #Stale.Q THEN
           #HaveSample := FALSE;
           IF #lastStatus = 0 THEN #lastStatus := DW#16#E0010003; END_IF;
       END_IF;
       IF NOT #Enable THEN #HaveSample := FALSE; END_IF;
       // Остаточна достовірність: придатний результат і чинний дозвіл опитування.
   #Valid := #HaveSample AND #Enable;
       IF NOT #Valid THEN #UpOrClosed := FALSE; #DownOrOpen := FALSE; END_IF;
       #Busy := #readBusy;
       #Status := #lastStatus;
END_FUNCTION_BLOCK

FUNCTION_BLOCK "FB_Diagnostics_Messages"   // FB621, LAD
{ S7_Optimized_Access := 'TRUE' }
VERSION : 0.1
   VAR
      ssfbHMI_w1 : "FB_DigIn_16_XOR";
      ssfbHMI_w2 : "FB_DigIn_16_XOR";
   END_VAR
BEGIN

